Staubli VAL3: Rect10.dtx

public frame fReference = {x=1475.172, y=-187.34, z=-1030, rz=81.293, fatherId=world[0]}
public jointRx jPark = {j3=90, j5=90}
public jointRx jJoint = {j1=-21.01263, j2=66.00245, j3=79.88662, j5=34.11093, j6=162.86516}
public mdesc mNomSpeed = {blend=off}
public mdesc mSpeed[30]
  [0] = {tmax=75, rmax=100, leave=0.1, reach=0.1, blend=cartesian}
  [1] = {tmax=75, rmax=100, leave=0.1, reach=0.1, blend=cartesian}
  [2] = {tmax=75, rmax=100, leave=0.1, reach=0.1, blend=cartesian}
  [3] = {tmax=75, rmax=100, leave=0.1, reach=0.1, blend=cartesian}
  [4] = {tmax=75, rmax=100, leave=0.1, reach=0.1, blend=cartesian}
  [5] = {tmax=75, rmax=100, leave=0.1, reach=0.1, blend=cartesian}
  [6] = {tmax=75, rmax=100, leave=0.1, reach=0.1, blend=cartesian}
  [7] = {tmax=75, rmax=100, leave=0.1, reach=0.1, blend=cartesian}
  [8] = {tmax=75, rmax=100, leave=0.1, reach=0.1, blend=cartesian}
  [9] = {tmax=75, rmax=100, leave=0.1, reach=0.1, blend=cartesian}
  [10] = {tmax=75, rmax=100, leave=0.1, reach=0.1, blend=cartesian}
  [11] = {tmax=75, rmax=100, leave=0.1, reach=0.1, blend=cartesian}
  [12] = {tmax=75, rmax=100, leave=0.1, reach=0.1, blend=cartesian}
  [13] = {tmax=75, rmax=100, leave=0.1, reach=0.1, blend=cartesian}
  [14] = {tmax=75, rmax=100, leave=0.1, reach=0.1, blend=cartesian}
  [15] = {tmax=75, rmax=100, leave=0.1, reach=0.1, blend=cartesian}
  [16] = {tmax=75, rmax=100, leave=0.1, reach=0.1, blend=cartesian}
  [17] = {tmax=75, rmax=100, leave=0.1, reach=0.1, blend=cartesian}
  [18] = {tmax=75, rmax=100, leave=0.1, reach=0.1, blend=cartesian}
  [19] = {tmax=75, rmax=100, leave=0.1, reach=0.1, blend=cartesian}
  [20] = {tmax=75, rmax=100, leave=0.1, reach=0.1, blend=cartesian}
  [21] = {tmax=75, rmax=100, leave=0.1, reach=0.1, blend=cartesian}
  [22] = {tmax=75, rmax=100, leave=0.1, reach=0.1, blend=cartesian}
  [23] = {tmax=75, rmax=100, leave=0.1, reach=0.1, blend=cartesian}
  [24] = {tmax=75, rmax=100, leave=0.1, reach=0.1, blend=cartesian}
  [25] = {tmax=75, rmax=100, leave=0.1, reach=0.1, blend=cartesian}
  [26] = {tmax=75, rmax=100, leave=0.1, reach=0.1, blend=cartesian}
  [27] = {tmax=75, rmax=100, leave=0.1, reach=0.1, blend=cartesian}
  [28] = {tmax=75, rmax=100, leave=0.1, reach=0.1, blend=cartesian}
  [29] = {tmax=75, rmax=100, leave=0.1, reach=0.1, blend=cartesian}
public num nTraj
num nTimeStop
num nTimeStart
num nMode
num nEtat
public pointRx pPoint[740]
  [0] = {x=-372, y=-44, z=100, rx=-180, rz=85.171, shoulder=lefty, elbow=epositive, wrist=wpositive, fatherId=fReference[0]}
  [1] = {x=-372, y=-44, rx=-180, rz=85.171, shoulder=lefty, elbow=epositive, wrist=wpositive, fatherId=fReference[0]}
  [2] = {x=-372, y=-44, rx=-180, rz=85.171, shoulder=lefty, elbow=epositive, wrist=wpositive, fatherId=fReference[0]}
  [3] = {x=-369.477, y=-73.864, rx=-180, rz=75.512, shoulder=lefty, elbow=epositive, wrist=wpositive, fatherId=fReference[0]}
  [4] = {x=-361.979, y=-102.881, rx=-180, rz=65.854, shoulder=lefty, elbow=epositive, wrist=wpositive, fatherId=fReference[0]}
  [5] = {x=-349.719, y=-130.229, rx=180, rz=56.195, shoulder=lefty, elbow=epositive, wrist=wpositive, fatherId=fReference[0]}
  [6] = {x=-333.045, y=-155.133, rx=-180, rz=46.537, shoulder=lefty, elbow=epositive, wrist=wpositive, fatherId=fReference[0]}
  [7] = {x=-312.429, y=-176.886, rx=-180, rz=36.878, shoulder=lefty, elbow=epositive, wrist=wpositive, fatherId=fReference[0]}
  [8] = {x=-288.455, y=-194.872, rx=180, rz=27.22, shoulder=lefty, elbow=epositive, wrist=wpositive, fatherId=fReference[0]}
  [9] = {x=-261.803, y=-208.58, rx=180, rz=17.561, shoulder=lefty, elbow=epositive, wrist=wpositive, fatherId=fReference[0]}
  [10] = {x=-233.23, y=-217.623, rx=180, rz=7.903, shoulder=lefty, elbow=epositive, wrist=wpositive, fatherId=fReference[0]}
  [11] = {x=-203.544, y=-221.744, rx=-180, rz=0.489, shoulder=lefty, elbow=epositive, wrist=wpositive, fatherId=fReference[0]}
  [12] = {x=-173.543, y=-222, rx=180, shoulder=lefty, elbow=epositive, wrist=wpositive, fatherId=fReference[0]}
  [13] = {x=-143.537, y=-222, rx=180, shoulder=lefty, elbow=epositive, wrist=wpositive, fatherId=fReference[0]}
  [14] = {x=-113.531, y=-222, rx=180, shoulder=lefty, elbow=epositive, wrist=wpositive, fatherId=fReference[0]}
  [15] = {x=-83.525, y=-222, rx=180, shoulder=lefty, elbow=epositive, wrist=wpositive, fatherId=fReference[0]}
  [16] = {x=-53.519, y=-222, rx=180, shoulder=lefty, elbow=epositive, wrist=wpositive, fatherId=fReference[0]}
  [17] = {x=-23.513, y=-222, rx=-180, shoulder=lefty, elbow=epositive, wrist=wpositive, fatherId=fReference[0]}
  [18] = {x=6.493, y=-222, rx=-180, shoulder=lefty, elbow=epositive, wrist=wpositive, fatherId=fReference[0]}
  [19] = {x=36.499, y=-222, rx=-180, shoulder=lefty, elbow=epositive, wrist=wpositive, fatherId=fReference[0]}
  [20] = {x=66.504, y=-222, rx=-180, shoulder=lefty, elbow=epositive, wrist=wpositive, fatherId=fReference[0]}
  [21] = {x=96.51, y=-222, rx=180, shoulder=lefty, elbow=epositive, wrist=wpositive, fatherId=fReference[0]}
  [22] = {x=126.516, y=-222, rx=180, shoulder=lefty, elbow=epositive, wrist=wpositive, fatherId=fReference[0]}
  [23] = {x=156.522, y=-222, rx=180, shoulder=lefty, elbow=epositive, wrist=wpositive, fatherId=fReference[0]}
  [24] = {x=186.528, y=-222, rx=-180, rz=-2.723, shoulder=lefty, elbow=epositive, wrist=wpositive, fatherId=fReference[0]}
  [25] = {x=216.474, y=-220.576, rx=180, rz=-12.083, shoulder=lefty, elbow=epositive, wrist=wpositive, fatherId=fReference[0]}
  [26] = {x=245.78, y=-214.302, rx=180, rz=-21.741, shoulder=lefty, elbow=epositive, wrist=wpositive, fatherId=fReference[0]}
  [27] = {x=273.619, y=-203.201, rx=180, rz=-31.4, shoulder=lefty, elbow=epositive, wrist=wpositive, fatherId=fReference[0]}
  [28] = {x=299.2, y=-187.586, rx=180, rz=-41.058, shoulder=lefty, elbow=epositive, wrist=wpositive, fatherId=fReference[0]}
  [29] = {x=321.799, y=-167.901, rx=-180, rz=-50.717, shoulder=lefty, elbow=epositive, wrist=wpositive, fatherId=fReference[0]}
  [30] = {x=340.775, y=-144.703, rx=-180, rz=-60.375, shoulder=lefty, elbow=epositive, wrist=wpositive, fatherId=fReference[0]}
  [31] = {x=355.59, y=-118.65, rx=180, rz=-70.034, shoulder=lefty, elbow=epositive, wrist=wpositive, fatherId=fReference[0]}
  [32] = {x=365.824, y=-90.481, rx=180, rz=-79.692, shoulder=lefty, elbow=epositive, wrist=wpositive, fatherId=fReference[0]}
  [33] = {x=371.187, y=-60.995, rx=180, rz=-88.446, shoulder=lefty, elbow=epositive, wrist=wpositive, fatherId=fReference[0]}
  [34] = {x=372, y=-31.015, rx=180, rz=-90, shoulder=lefty, elbow=epositive, wrist=wpositive, fatherId=fReference[0]}
  [35] = {x=372, y=-1.009, rx=180, rz=-90, shoulder=lefty, elbow=epositive, wrist=wpositive, fatherId=fReference[0]}
  [36] = {x=372, y=28.997, rx=-180, rz=-91.207, shoulder=lefty, elbow=epositive, wrist=wpositive, fatherId=fReference[0]}
  [37] = {x=371.368, y=58.985, rx=-180, rz=-99.658, shoulder=lefty, elbow=epositive, wrist=wpositive, fatherId=fReference[0]}
  [38] = {x=366.34, y=88.531, rx=-180, rz=-109.317, shoulder=lefty, elbow=epositive, wrist=wpositive, fatherId=fReference[0]}
  [39] = {x=356.426, y=116.814, rx=-180, rz=-118.975, shoulder=lefty, elbow=epositive, wrist=wpositive, fatherId=fReference[0]}
  [40] = {x=341.907, y=143.033, rx=-180, rz=-128.634, shoulder=lefty, elbow=epositive, wrist=wpositive, fatherId=fReference[0]}
  [41] = {x=323.195, y=166.444, rx=-180, rz=-138.292, shoulder=lefty, elbow=epositive, wrist=wpositive, fatherId=fReference[0]}
  [42] = {x=300.821, y=186.384, rx=180, rz=-147.951, shoulder=lefty, elbow=epositive, wrist=wpositive, fatherId=fReference[0]}
  [43] = {x=275.418, y=202.288, rx=-180, rz=-157.609, shoulder=lefty, elbow=epositive, wrist=wpositive, fatherId=fReference[0]}
  [44] = {x=247.707, y=213.704, rx=-180, rz=-167.268, shoulder=lefty, elbow=epositive, wrist=wpositive, fatherId=fReference[0]}
  [45] = {x=218.474, y=220.309, rx=-180, rz=-176.767, shoulder=lefty, elbow=epositive, wrist=wpositive, fatherId=fReference[0]}
  [46] = {x=188.546, y=222, rx=-180, rz=180, shoulder=lefty, elbow=epositive, wrist=wpositive, fatherId=fReference[0]}
  [47] = {x=158.54, y=222, rx=-180, rz=180, shoulder=lefty, elbow=epositive, wrist=wpositive, fatherId=fReference[0]}
  [48] = {x=128.534, y=222, rx=-180, rz=180, shoulder=lefty, elbow=epositive, wrist=wpositive, fatherId=fReference[0]}
  [49] = {x=98.528, y=222, rx=-180, rz=180, shoulder=lefty, elbow=epositive, wrist=wpositive, fatherId=fReference[0]}
  [50] = {x=68.522, y=222, rx=-180, rz=180, shoulder=lefty, elbow=epositive, wrist=wpositive, fatherId=fReference[0]}
  [51] = {x=38.516, y=222, rx=-180, rz=180, shoulder=lefty, elbow=epositive, wrist=wpositive, fatherId=fReference[0]}
  [52] = {x=8.51, y=222, rx=-180, rz=180, shoulder=lefty, elbow=epositive, wrist=wpositive, fatherId=fReference[0]}
  [53] = {x=-21.496, y=222, rx=180, rz=180, shoulder=lefty, elbow=epositive, wrist=wpositive, fatherId=fReference[0]}
  [54] = {x=-51.501, y=222, rx=180, rz=180, shoulder=lefty, elbow=epositive, wrist=wpositive, fatherId=fReference[0]}
  [55] = {x=-81.507, y=222, rx=-180, rz=180, shoulder=lefty, elbow=epositive, wrist=wpositive, fatherId=fReference[0]}
  [56] = {x=-111.513, y=222, rx=-180, rz=180, shoulder=lefty, elbow=epositive, wrist=wpositive, fatherId=fReference[0]}
  [57] = {x=-141.519, y=222, rx=180, rz=180, shoulder=lefty, elbow=epositive, wrist=wpositive, fatherId=fReference[0]}
  [58] = {x=-171.525, y=222, rx=180, rz=179.696, shoulder=lefty, elbow=epositive, wrist=wpositive, fatherId=fReference[0]}
  [59] = {x=-201.529, y=221.841, rx=-180, rz=172.747, shoulder=lefty, elbow=epositive, wrist=wpositive, fatherId=fReference[0]}
  [60] = {x=-231.259, y=218.057, rx=-180, rz=163.088, shoulder=lefty, elbow=epositive, wrist=wpositive, fatherId=fReference[0]}
  [61] = {x=-259.934, y=209.338, rx=180, rz=153.43, shoulder=lefty, elbow=epositive, wrist=wpositive, fatherId=fReference[0]}
  [62] = {x=-286.739, y=195.933, rx=180, rz=143.771, shoulder=lefty, elbow=epositive, wrist=wpositive, fatherId=fReference[0]}
  [63] = {x=-310.915, y=178.22, rx=180, rz=134.113, shoulder=lefty, elbow=epositive, wrist=wpositive, fatherId=fReference[0]}
  [64] = {x=-331.776, y=156.702, rx=180, rz=124.454, shoulder=lefty, elbow=epositive, wrist=wpositive, fatherId=fReference[0]}
  [65] = {x=-348.732, y=131.989, rx=180, rz=114.796, shoulder=lefty, elbow=epositive, wrist=wpositive, fatherId=fReference[0]}
  [66] = {x=-361.301, y=104.782, rx=180, rz=105.137, shoulder=lefty, elbow=epositive, wrist=wpositive, fatherId=fReference[0]}
  [67] = {x=-369.127, y=75.851, rx=180, rz=95.479, shoulder=lefty, elbow=epositive, wrist=wpositive, fatherId=fReference[0]}
  [68] = {x=-371.989, y=46.018, rx=180, rz=90.022, shoulder=lefty, elbow=epositive, wrist=wpositive, fatherId=fReference[0]}
  [69] = {x=-372, y=16.012, rx=-180, rz=90, shoulder=lefty, elbow=epositive, wrist=wpositive, fatherId=fReference[0]}
  [70] = {x=-372, y=-13.994, rx=-180, rz=90, shoulder=lefty, elbow=epositive, wrist=wpositive, fatherId=fReference[0]}
  [71] = {x=-372, y=-44, rx=-180, rz=90, shoulder=lefty, elbow=epositive, wrist=wpositive, fatherId=fReference[0]}
  [72] = {x=-372, y=-44, rx=-180, rz=90, shoulder=lefty, elbow=epositive, wrist=wpositive, fatherId=fReference[0]}
  [73] = {x=-372, y=-44, z=100, rx=-180, rz=90, shoulder=lefty, elbow=epositive, wrist=wpositive, fatherId=fReference[0]}
  [74] = {x=-372, y=-44, z=122, rx=-180, rz=90, shoulder=lefty, elbow=epositive, wrist=wpositive, fatherId=fReference[0]}
  [75] = {x=-372, y=-44, z=22, rx=-180, rz=90, shoulder=lefty, elbow=epositive, wrist=wpositive, fatherId=fReference[0]}
  [76] = {x=-372, y=-44, z=22, rx=-180, rz=90, shoulder=lefty, elbow=epositive, wrist=wpositive, fatherId=fReference[0]}
  [77] = {x=-372, y=-13.994, z=22, rx=-180, rz=90, shoulder=lefty, elbow=epositive, wrist=wpositive, fatherId=fReference[0]}
  [78] = {x=-372, y=16.012, z=22, rx=180, rz=90.022, shoulder=lefty, elbow=epositive, wrist=wpositive, fatherId=fReference[0]}
  [79] = {x=-371.989, y=46.018, z=22, rx=180, rz=95.479, shoulder=lefty, elbow=epositive, wrist=wpositive, fatherId=fReference[0]}
  [80] = {x=-369.127, y=75.851, z=22, rx=180, rz=105.137, shoulder=lefty, elbow=epositive, wrist=wpositive, fatherId=fReference[0]}
  [81] = {x=-361.301, y=104.782, z=22, rx=180, rz=114.796, shoulder=lefty, elbow=epositive, wrist=wpositive, fatherId=fReference[0]}
  [82] = {x=-348.732, y=131.989, z=22, rx=180, rz=124.454, shoulder=lefty, elbow=epositive, wrist=wpositive, fatherId=fReference[0]}
  [83] = {x=-331.776, y=156.702, z=22, rx=180, rz=134.113, shoulder=lefty, elbow=epositive, wrist=wpositive, fatherId=fReference[0]}
  [84] = {x=-310.915, y=178.22, z=22, rx=180, rz=143.771, shoulder=lefty, elbow=epositive, wrist=wpositive, fatherId=fReference[0]}
  [85] = {x=-286.739, y=195.933, z=22, rx=180, rz=153.43, shoulder=lefty, elbow=epositive, wrist=wpositive, fatherId=fReference[0]}
  [86] = {x=-259.934, y=209.338, z=22, rx=180, rz=163.088, shoulder=lefty, elbow=epositive, wrist=wpositive, fatherId=fReference[0]}
  [87] = {x=-231.259, y=218.057, z=22, rx=-180, rz=172.747, shoulder=lefty, elbow=epositive, wrist=wpositive, fatherId=fReference[0]}
  [88] = {x=-201.529, y=221.841, z=22, rx=180, rz=179.696, shoulder=lefty, elbow=epositive, wrist=wpositive, fatherId=fReference[0]}
  [89] = {x=-171.525, y=222, z=22, rx=180, rz=180, shoulder=lefty, elbow=epositive, wrist=wpositive, fatherId=fReference[0]}
  [90] = {x=-141.519, y=222, z=22, rx=-180, rz=180, shoulder=lefty, elbow=epositive, wrist=wpositive, fatherId=fReference[0]}
  [91] = {x=-111.513, y=222, z=22, rx=180, rz=180, shoulder=lefty, elbow=epositive, wrist=wpositive, fatherId=fReference[0]}
  [92] = {x=-81.507, y=222, z=22, rx=-180, rz=180, shoulder=lefty, elbow=epositive, wrist=wpositive, fatherId=fReference[0]}
  [93] = {x=-51.501, y=222, z=22, rx=180, rz=180, shoulder=lefty, elbow=epositive, wrist=wpositive, fatherId=fReference[0]}
  [94] = {x=-21.496, y=222, z=22, rx=180, rz=180, shoulder=lefty, elbow=epositive, wrist=wpositive, fatherId=fReference[0]}
  [95] = {x=8.51, y=222, z=22, rx=-180, rz=180, shoulder=lefty, elbow=epositive, wrist=wpositive, fatherId=fReference[0]}
  [96] = {x=38.516, y=222, z=22, rx=180, rz=180, shoulder=lefty, elbow=epositive, wrist=wpositive, fatherId=fReference[0]}
  [97] = {x=68.522, y=222, z=22, rx=180, rz=180, shoulder=lefty, elbow=epositive, wrist=wpositive, fatherId=fReference[0]}
  [98] = {x=98.528, y=222, z=22, rx=-180, rz=180, shoulder=lefty, elbow=epositive, wrist=wpositive, fatherId=fReference[0]}
  [99] = {x=128.534, y=222, z=22, rx=180, rz=180, shoulder=lefty, elbow=epositive, wrist=wpositive, fatherId=fReference[0]}
  [100] = {x=158.54, y=222, z=22, rx=180, rz=180, shoulder=lefty, elbow=epositive, wrist=wpositive, fatherId=fReference[0]}
  [101] = {x=188.546, y=222, z=22, rx=-180, rz=-176.767, shoulder=lefty, elbow=epositive, wrist=wpositive, fatherId=fReference[0]}
  [102] = {x=218.474, y=220.309, z=22, rx=180, rz=-167.268, shoulder=lefty, elbow=epositive, wrist=wpositive, fatherId=fReference[0]}
  [103] = {x=247.707, y=213.704, z=22, rx=-180, rz=-157.609, shoulder=lefty, elbow=epositive, wrist=wpositive, fatherId=fReference[0]}
  [104] = {x=275.418, y=202.288, z=22, rx=180, rz=-147.951, shoulder=lefty, elbow=epositive, wrist=wpositive, fatherId=fReference[0]}
  [105] = {x=300.821, y=186.384, z=22, rx=-180, rz=-138.292, shoulder=lefty, elbow=epositive, wrist=wpositive, fatherId=fReference[0]}
  [106] = {x=323.195, y=166.444, z=22, rx=-180, rz=-128.634, shoulder=lefty, elbow=epositive, wrist=wpositive, fatherId=fReference[0]}
  [107] = {x=341.907, y=143.033, z=22, rx=-180, rz=-118.975, shoulder=lefty, elbow=epositive, wrist=wpositive, fatherId=fReference[0]}
  [108] = {x=356.426, y=116.814, z=22, rx=-180, rz=-109.317, shoulder=lefty, elbow=epositive, wrist=wpositive, fatherId=fReference[0]}
  [109] = {x=366.34, y=88.531, z=22, rx=-180, rz=-99.658, shoulder=lefty, elbow=epositive, wrist=wpositive, fatherId=fReference[0]}
  [110] = {x=371.368, y=58.985, z=22, rx=-180, rz=-91.207, shoulder=lefty, elbow=epositive, wrist=wpositive, fatherId=fReference[0]}
  [111] = {x=372, y=28.997, z=22, rx=180, rz=-90, shoulder=lefty, elbow=epositive, wrist=wpositive, fatherId=fReference[0]}
  [112] = {x=372, y=-1.009, z=22, rx=180, rz=-90, shoulder=lefty, elbow=epositive, wrist=wpositive, fatherId=fReference[0]}
  [113] = {x=372, y=-31.015, z=22, rx=180, rz=-88.446, shoulder=lefty, elbow=epositive, wrist=wpositive, fatherId=fReference[0]}
  [114] = {x=371.187, y=-60.995, z=22, rx=180, rz=-79.692, shoulder=lefty, elbow=epositive, wrist=wpositive, fatherId=fReference[0]}
  [115] = {x=365.824, y=-90.481, z=22, rx=180, rz=-70.034, shoulder=lefty, elbow=epositive, wrist=wpositive, fatherId=fReference[0]}
  [116] = {x=355.59, y=-118.65, z=22, rx=-180, rz=-60.375, shoulder=lefty, elbow=epositive, wrist=wpositive, fatherId=fReference[0]}
  [117] = {x=340.775, y=-144.703, z=22, rx=180, rz=-50.717, shoulder=lefty, elbow=epositive, wrist=wpositive, fatherId=fReference[0]}
  [118] = {x=321.799, y=-167.901, z=22, rx=180, rz=-41.058, shoulder=lefty, elbow=epositive, wrist=wpositive, fatherId=fReference[0]}
  [119] = {x=299.2, y=-187.586, z=22, rx=180, rz=-31.4, shoulder=lefty, elbow=epositive, wrist=wpositive, fatherId=fReference[0]}
  [120] = {x=273.619, y=-203.201, z=22, rx=180, rz=-21.741, shoulder=lefty, elbow=epositive, wrist=wpositive, fatherId=fReference[0]}
  [121] = {x=245.78, y=-214.302, z=22, rx=180, rz=-12.083, shoulder=lefty, elbow=epositive, wrist=wpositive, fatherId=fReference[0]}
  [122] = {x=216.474, y=-220.576, z=22, rx=-180, rz=-2.723, shoulder=lefty, elbow=epositive, wrist=wpositive, fatherId=fReference[0]}
  [123] = {x=186.528, y=-222, z=22, rx=-180, shoulder=lefty, elbow=epositive, wrist=wpositive, fatherId=fReference[0]}
  [124] = {x=156.522, y=-222, z=22, rx=-180, shoulder=lefty, elbow=epositive, wrist=wpositive, fatherId=fReference[0]}
  [125] = {x=126.516, y=-222, z=22, rx=-180, shoulder=lefty, elbow=epositive, wrist=wpositive, fatherId=fReference[0]}
  [126] = {x=96.51, y=-222, z=22, rx=-180, shoulder=lefty, elbow=epositive, wrist=wpositive, fatherId=fReference[0]}
  [127] = {x=66.504, y=-222, z=22, rx=-180, shoulder=lefty, elbow=epositive, wrist=wpositive, fatherId=fReference[0]}
  [128] = {x=36.499, y=-222, z=22, rx=-180, shoulder=lefty, elbow=epositive, wrist=wpositive, fatherId=fReference[0]}
  [129] = {x=6.493, y=-222, z=22, rx=-180, shoulder=lefty, elbow=epositive, wrist=wpositive, fatherId=fReference[0]}
  [130] = {x=-23.513, y=-222, z=22, rx=180, shoulder=lefty, elbow=epositive, wrist=wpositive, fatherId=fReference[0]}
  [131] = {x=-53.519, y=-222, z=22, rx=180, shoulder=lefty, elbow=epositive, wrist=wpositive, fatherId=fReference[0]}
  [132] = {x=-83.525, y=-222, z=22, rx=-180, shoulder=lefty, elbow=epositive, wrist=wpositive, fatherId=fReference[0]}
  [133] = {x=-113.531, y=-222, z=22, rx=180, shoulder=lefty, elbow=epositive, wrist=wpositive, fatherId=fReference[0]}
  [134] = {x=-143.537, y=-222, z=22, rx=-180, shoulder=lefty, elbow=epositive, wrist=wpositive, fatherId=fReference[0]}
  [135] = {x=-173.543, y=-222, z=22, rx=180, rz=0.489, shoulder=lefty, elbow=epositive, wrist=wpositive, fatherId=fReference[0]}
  [136] = {x=-203.544, y=-221.744, z=22, rx=180, rz=7.903, shoulder=lefty, elbow=epositive, wrist=wpositive, fatherId=fReference[0]}
  [137] = {x=-233.23, y=-217.623, z=22, rx=-180, rz=17.561, shoulder=lefty, elbow=epositive, wrist=wpositive, fatherId=fReference[0]}
  [138] = {x=-261.803, y=-208.58, z=22, rx=-180, rz=27.22, shoulder=lefty, elbow=epositive, wrist=wpositive, fatherId=fReference[0]}
  [139] = {x=-288.455, y=-194.872, z=22, rx=-180, rz=36.878, shoulder=lefty, elbow=epositive, wrist=wpositive, fatherId=fReference[0]}
  [140] = {x=-312.429, y=-176.886, z=22, rx=-180, rz=46.537, shoulder=lefty, elbow=epositive, wrist=wpositive, fatherId=fReference[0]}
  [141] = {x=-333.045, y=-155.133, z=22, rx=-180, rz=56.195, shoulder=lefty, elbow=epositive, wrist=wpositive, fatherId=fReference[0]}
  [142] = {x=-349.719, y=-130.229, z=22, rx=180, rz=65.854, shoulder=lefty, elbow=epositive, wrist=wpositive, fatherId=fReference[0]}
  [143] = {x=-361.979, y=-102.881, z=22, rx=-180, rz=75.512, shoulder=lefty, elbow=epositive, wrist=wpositive, fatherId=fReference[0]}
  [144] = {x=-369.477, y=-73.864, z=22, rx=-180, rz=85.171, shoulder=lefty, elbow=epositive, wrist=wpositive, fatherId=fReference[0]}
  [145] = {x=-372, y=-44, z=22, rx=-180, rz=85.171, shoulder=lefty, elbow=epositive, wrist=wpositive, fatherId=fReference[0]}
  [146] = {x=-372, y=-44, z=22, rx=-180, rz=85.171, shoulder=lefty, elbow=epositive, wrist=wpositive, fatherId=fReference[0]}
  [147] = {x=-372, y=-44, z=122, rx=-180, rz=85.171, shoulder=lefty, elbow=epositive, wrist=wpositive, fatherId=fReference[0]}
  [148] = {x=-372, y=-44, z=144, rx=-180, rz=85.171, shoulder=lefty, elbow=epositive, wrist=wpositive, fatherId=fReference[0]}
  [149] = {x=-372, y=-44, z=44, rx=-180, rz=85.171, shoulder=lefty, elbow=epositive, wrist=wpositive, fatherId=fReference[0]}
  [150] = {x=-372, y=-44, z=44, rx=-180, rz=85.171, shoulder=lefty, elbow=epositive, wrist=wpositive, fatherId=fReference[0]}
  [151] = {x=-369.477, y=-73.864, z=44, rx=-180, rz=75.512, shoulder=lefty, elbow=epositive, wrist=wpositive, fatherId=fReference[0]}
  [152] = {x=-361.979, y=-102.881, z=44, rx=-180, rz=65.854, shoulder=lefty, elbow=epositive, wrist=wpositive, fatherId=fReference[0]}
  [153] = {x=-349.719, y=-130.229, z=44, rx=-180, rz=56.195, shoulder=lefty, elbow=epositive, wrist=wpositive, fatherId=fReference[0]}
  [154] = {x=-333.045, y=-155.133, z=44, rx=180, rz=46.537, shoulder=lefty, elbow=epositive, wrist=wpositive, fatherId=fReference[0]}
  [155] = {x=-312.429, y=-176.886, z=44, rx=-180, rz=36.878, shoulder=lefty, elbow=epositive, wrist=wpositive, fatherId=fReference[0]}
  [156] = {x=-288.455, y=-194.872, z=44, rx=180, rz=27.22, shoulder=lefty, elbow=epositive, wrist=wpositive, fatherId=fReference[0]}
  [157] = {x=-261.803, y=-208.58, z=44, rx=-180, rz=17.561, shoulder=lefty, elbow=epositive, wrist=wpositive, fatherId=fReference[0]}
  [158] = {x=-233.23, y=-217.623, z=44, rx=-180, rz=7.903, shoulder=lefty, elbow=epositive, wrist=wpositive, fatherId=fReference[0]}
  [159] = {x=-203.544, y=-221.744, z=44, rx=-180, rz=0.489, shoulder=lefty, elbow=epositive, wrist=wpositive, fatherId=fReference[0]}
  [160] = {x=-173.543, y=-222, z=44, rx=-180, shoulder=lefty, elbow=epositive, wrist=wpositive, fatherId=fReference[0]}
  [161] = {x=-143.537, y=-222, z=44, rx=180, shoulder=lefty, elbow=epositive, wrist=wpositive, fatherId=fReference[0]}
  [162] = {x=-113.531, y=-222, z=44, rx=180, shoulder=lefty, elbow=epositive, wrist=wpositive, fatherId=fReference[0]}
  [163] = {x=-83.525, y=-222, z=44, rx=-180, shoulder=lefty, elbow=epositive, wrist=wpositive, fatherId=fReference[0]}
  [164] = {x=-53.519, y=-222, z=44, rx=180, shoulder=lefty, elbow=epositive, wrist=wpositive, fatherId=fReference[0]}
  [165] = {x=-23.513, y=-222, z=44, rx=180, shoulder=lefty, elbow=epositive, wrist=wpositive, fatherId=fReference[0]}
  [166] = {x=6.493, y=-222, z=44, rx=180, shoulder=lefty, elbow=epositive, wrist=wpositive, fatherId=fReference[0]}
  [167] = {x=36.499, y=-222, z=44, rx=-180, shoulder=lefty, elbow=epositive, wrist=wpositive, fatherId=fReference[0]}
  [168] = {x=66.504, y=-222, z=44, rx=-180, shoulder=lefty, elbow=epositive, wrist=wpositive, fatherId=fReference[0]}
  [169] = {x=96.51, y=-222, z=44, rx=-180, shoulder=lefty, elbow=epositive, wrist=wpositive, fatherId=fReference[0]}
  [170] = {x=126.516, y=-222, z=44, rx=-180, shoulder=lefty, elbow=epositive, wrist=wpositive, fatherId=fReference[0]}
  [171] = {x=156.522, y=-222, z=44, rx=180, shoulder=lefty, elbow=epositive, wrist=wpositive, fatherId=fReference[0]}
  [172] = {x=186.528, y=-222, z=44, rx=-180, rz=-2.723, shoulder=lefty, elbow=epositive, wrist=wpositive, fatherId=fReference[0]}
  [173] = {x=216.474, y=-220.576, z=44, rx=-180, rz=-12.083, shoulder=lefty, elbow=epositive, wrist=wpositive, fatherId=fReference[0]}
  [174] = {x=245.78, y=-214.302, z=44, rx=180, rz=-21.741, shoulder=lefty, elbow=epositive, wrist=wpositive, fatherId=fReference[0]}
  [175] = {x=273.619, y=-203.201, z=44, rx=180, rz=-31.4, shoulder=lefty, elbow=epositive, wrist=wpositive, fatherId=fReference[0]}
  [176] = {x=299.2, y=-187.586, z=44, rx=180, rz=-41.058, shoulder=lefty, elbow=epositive, wrist=wpositive, fatherId=fReference[0]}
  [177] = {x=321.799, y=-167.901, z=44, rx=180, rz=-50.717, shoulder=lefty, elbow=epositive, wrist=wpositive, fatherId=fReference[0]}
  [178] = {x=340.775, y=-144.703, z=44, rx=180, rz=-60.375, shoulder=lefty, elbow=epositive, wrist=wpositive, fatherId=fReference[0]}
  [179] = {x=355.59, y=-118.65, z=44, rx=-180, rz=-70.034, shoulder=lefty, elbow=epositive, wrist=wpositive, fatherId=fReference[0]}
  [180] = {x=365.824, y=-90.481, z=44, rx=180, rz=-79.692, shoulder=lefty, elbow=epositive, wrist=wpositive, fatherId=fReference[0]}
  [181] = {x=371.187, y=-60.995, z=44, rx=180, rz=-88.446, shoulder=lefty, elbow=epositive, wrist=wpositive, fatherId=fReference[0]}
  [182] = {x=372, y=-31.015, z=44, rx=180, rz=-90, shoulder=lefty, elbow=epositive, wrist=wpositive, fatherId=fReference[0]}
  [183] = {x=372, y=-1.009, z=44, rx=180, rz=-90, shoulder=lefty, elbow=epositive, wrist=wpositive, fatherId=fReference[0]}
  [184] = {x=372, y=28.997, z=44, rx=-180, rz=-91.207, shoulder=lefty, elbow=epositive, wrist=wpositive, fatherId=fReference[0]}
  [185] = {x=371.368, y=58.985, z=44, rx=-180, rz=-99.658, shoulder=lefty, elbow=epositive, wrist=wpositive, fatherId=fReference[0]}
  [186] = {x=366.34, y=88.531, z=44, rx=-180, rz=-109.317, shoulder=lefty, elbow=epositive, wrist=wpositive, fatherId=fReference[0]}
  [187] = {x=356.426, y=116.814, z=44, rx=-180, rz=-118.975, shoulder=lefty, elbow=epositive, wrist=wpositive, fatherId=fReference[0]}
  [188] = {x=341.907, y=143.033, z=44, rx=-180, rz=-128.634, shoulder=lefty, elbow=epositive, wrist=wpositive, fatherId=fReference[0]}
  [189] = {x=323.195, y=166.444, z=44, rx=-180, rz=-138.292, shoulder=lefty, elbow=epositive, wrist=wpositive, fatherId=fReference[0]}
  [190] = {x=300.821, y=186.384, z=44, rx=-180, rz=-147.951, shoulder=lefty, elbow=epositive, wrist=wpositive, fatherId=fReference[0]}
  [191] = {x=275.418, y=202.288, z=44, rx=180, rz=-157.609, shoulder=lefty, elbow=epositive, wrist=wpositive, fatherId=fReference[0]}
  [192] = {x=247.707, y=213.704, z=44, rx=-180, rz=-167.268, shoulder=lefty, elbow=epositive, wrist=wpositive, fatherId=fReference[0]}
  [193] = {x=218.474, y=220.309, z=44, rx=-180, rz=-176.767, shoulder=lefty, elbow=epositive, wrist=wpositive, fatherId=fReference[0]}
  [194] = {x=188.546, y=222, z=44, rx=180, rz=180, shoulder=lefty, elbow=epositive, wrist=wpositive, fatherId=fReference[0]}
  [195] = {x=158.54, y=222, z=44, rx=-180, rz=180, shoulder=lefty, elbow=epositive, wrist=wpositive, fatherId=fReference[0]}
  [196] = {x=128.534, y=222, z=44, rx=-180, rz=180, shoulder=lefty, elbow=epositive, wrist=wpositive, fatherId=fReference[0]}
  [197] = {x=98.528, y=222, z=44, rx=180, rz=-180, shoulder=lefty, elbow=epositive, wrist=wpositive, fatherId=fReference[0]}
  [198] = {x=68.522, y=222, z=44, rx=180, rz=-180, shoulder=lefty, elbow=epositive, wrist=wpositive, fatherId=fReference[0]}
  [199] = {x=38.516, y=222, z=44, rx=180, rz=180, shoulder=lefty, elbow=epositive, wrist=wpositive, fatherId=fReference[0]}
  [200] = {x=8.51, y=222, z=44, rx=-180, rz=180, shoulder=lefty, elbow=epositive, wrist=wpositive, fatherId=fReference[0]}
  [201] = {x=-21.496, y=222, z=44, rx=180, rz=180, shoulder=lefty, elbow=epositive, wrist=wpositive, fatherId=fReference[0]}
  [202] = {x=-51.501, y=222, z=44, rx=180, rz=180, shoulder=lefty, elbow=epositive, wrist=wpositive, fatherId=fReference[0]}
  [203] = {x=-81.507, y=222, z=44, rx=-180, rz=180, shoulder=lefty, elbow=epositive, wrist=wpositive, fatherId=fReference[0]}
  [204] = {x=-111.513, y=222, z=44, rx=180, rz=-180, shoulder=lefty, elbow=epositive, wrist=wpositive, fatherId=fReference[0]}
  [205] = {x=-141.519, y=222, z=44, rx=-180, rz=-180, shoulder=lefty, elbow=epositive, wrist=wpositive, fatherId=fReference[0]}
  [206] = {x=-171.525, y=222, z=44, rx=180, rz=179.696, shoulder=lefty, elbow=epositive, wrist=wpositive, fatherId=fReference[0]}
  [207] = {x=-201.529, y=221.841, z=44, rx=-180, rz=172.747, shoulder=lefty, elbow=epositive, wrist=wpositive, fatherId=fReference[0]}
  [208] = {x=-231.259, y=218.057, z=44, rx=-180, rz=163.088, shoulder=lefty, elbow=epositive, wrist=wpositive, fatherId=fReference[0]}
  [209] = {x=-259.934, y=209.338, z=44, rx=-180, rz=153.43, shoulder=lefty, elbow=epositive, wrist=wpositive, fatherId=fReference[0]}
  [210] = {x=-286.739, y=195.933, z=44, rx=-180, rz=143.771, shoulder=lefty, elbow=epositive, wrist=wpositive, fatherId=fReference[0]}
  [211] = {x=-310.915, y=178.22, z=44, rx=180, rz=134.113, shoulder=lefty, elbow=epositive, wrist=wpositive, fatherId=fReference[0]}
  [212] = {x=-331.776, y=156.702, z=44, rx=180, rz=124.454, shoulder=lefty, elbow=epositive, wrist=wpositive, fatherId=fReference[0]}
  [213] = {x=-348.732, y=131.989, z=44, rx=180, rz=114.796, shoulder=lefty, elbow=epositive, wrist=wpositive, fatherId=fReference[0]}
  [214] = {x=-361.301, y=104.782, z=44, rx=180, rz=105.137, shoulder=lefty, elbow=epositive, wrist=wpositive, fatherId=fReference[0]}
  [215] = {x=-369.127, y=75.851, z=44, rx=180, rz=95.479, shoulder=lefty, elbow=epositive, wrist=wpositive, fatherId=fReference[0]}
  [216] = {x=-371.989, y=46.018, z=44, rx=180, rz=90.022, shoulder=lefty, elbow=epositive, wrist=wpositive, fatherId=fReference[0]}
  [217] = {x=-372, y=16.012, z=44, rx=-180, rz=90, shoulder=lefty, elbow=epositive, wrist=wpositive, fatherId=fReference[0]}
  [218] = {x=-372, y=-13.994, z=44, rx=-180, rz=90, shoulder=lefty, elbow=epositive, wrist=wpositive, fatherId=fReference[0]}
  [219] = {x=-372, y=-44, z=44, rx=-180, rz=90, shoulder=lefty, elbow=epositive, wrist=wpositive, fatherId=fReference[0]}
  [220] = {x=-372, y=-44, z=44, rx=-180, rz=90, shoulder=lefty, elbow=epositive, wrist=wpositive, fatherId=fReference[0]}
  [221] = {x=-372, y=-44, z=144, rx=-180, rz=90, shoulder=lefty, elbow=epositive, wrist=wpositive, fatherId=fReference[0]}
  [222] = {x=-372, y=-44, z=166, rx=-180, rz=90, shoulder=lefty, elbow=epositive, wrist=wpositive, fatherId=fReference[0]}
  [223] = {x=-372, y=-44, z=66, rx=-180, rz=90, shoulder=lefty, elbow=epositive, wrist=wpositive, fatherId=fReference[0]}
  [224] = {x=-372, y=-44, z=66, rx=-180, rz=90, shoulder=lefty, elbow=epositive, wrist=wpositive, fatherId=fReference[0]}
  [225] = {x=-372, y=-13.994, z=66, rx=-180, rz=90, shoulder=lefty, elbow=epositive, wrist=wpositive, fatherId=fReference[0]}
  [226] = {x=-372, y=16.012, z=66, rx=180, rz=90.022, shoulder=lefty, elbow=epositive, wrist=wpositive, fatherId=fReference[0]}
  [227] = {x=-371.989, y=46.018, z=66, rx=180, rz=95.479, shoulder=lefty, elbow=epositive, wrist=wpositive, fatherId=fReference[0]}
  [228] = {x=-369.127, y=75.851, z=66, rx=180, rz=105.137, shoulder=lefty, elbow=epositive, wrist=wpositive, fatherId=fReference[0]}
  [229] = {x=-361.301, y=104.782, z=66, rx=180, rz=114.796, shoulder=lefty, elbow=epositive, wrist=wpositive, fatherId=fReference[0]}
  [230] = {x=-348.732, y=131.989, z=66, rx=180, rz=124.454, shoulder=lefty, elbow=epositive, wrist=wpositive, fatherId=fReference[0]}
  [231] = {x=-331.776, y=156.702, z=66, rx=180, rz=134.113, shoulder=lefty, elbow=epositive, wrist=wpositive, fatherId=fReference[0]}
  [232] = {x=-310.915, y=178.22, z=66, rx=-180, rz=143.771, shoulder=lefty, elbow=epositive, wrist=wpositive, fatherId=fReference[0]}
  [233] = {x=-286.739, y=195.933, z=66, rx=180, rz=153.43, shoulder=lefty, elbow=epositive, wrist=wpositive, fatherId=fReference[0]}
  [234] = {x=-259.934, y=209.338, z=66, rx=180, rz=163.088, shoulder=lefty, elbow=epositive, wrist=wpositive, fatherId=fReference[0]}
  [235] = {x=-231.259, y=218.057, z=66, rx=180, rz=172.747, shoulder=lefty, elbow=epositive, wrist=wpositive, fatherId=fReference[0]}
  [236] = {x=-201.529, y=221.841, z=66, rx=-180, rz=179.696, shoulder=lefty, elbow=epositive, wrist=wpositive, fatherId=fReference[0]}
  [237] = {x=-171.525, y=222, z=66, rx=-180, rz=180, shoulder=lefty, elbow=epositive, wrist=wpositive, fatherId=fReference[0]}
  [238] = {x=-141.519, y=222, z=66, rx=180, rz=-180, shoulder=lefty, elbow=epositive, wrist=wpositive, fatherId=fReference[0]}
  [239] = {x=-111.513, y=222, z=66, rx=180, rz=-180, shoulder=lefty, elbow=epositive, wrist=wpositive, fatherId=fReference[0]}
  [240] = {x=-81.507, y=222, z=66, rx=-180, rz=-180, shoulder=lefty, elbow=epositive, wrist=wpositive, fatherId=fReference[0]}
  [241] = {x=-51.501, y=222, z=66, rx=180, rz=180, shoulder=lefty, elbow=epositive, wrist=wpositive, fatherId=fReference[0]}
  [242] = {x=-21.496, y=222, z=66, rx=180, rz=-180, shoulder=lefty, elbow=epositive, wrist=wpositive, fatherId=fReference[0]}
  [243] = {x=8.51, y=222, z=66, rx=-180, rz=-180, shoulder=lefty, elbow=epositive, wrist=wpositive, fatherId=fReference[0]}
  [244] = {x=38.516, y=222, z=66, rx=-180, rz=-180, shoulder=lefty, elbow=epositive, wrist=wpositive, fatherId=fReference[0]}
  [245] = {x=68.522, y=222, z=66, rx=-180, rz=-180, shoulder=lefty, elbow=epositive, wrist=wpositive, fatherId=fReference[0]}
  [246] = {x=98.528, y=222, z=66, rx=180, rz=-180, shoulder=lefty, elbow=epositive, wrist=wpositive, fatherId=fReference[0]}
  [247] = {x=128.534, y=222, z=66, rx=180, rz=180, shoulder=lefty, elbow=epositive, wrist=wpositive, fatherId=fReference[0]}
  [248] = {x=158.54, y=222, z=66, rx=180, rz=-180, shoulder=lefty, elbow=epositive, wrist=wpositive, fatherId=fReference[0]}
  [249] = {x=188.546, y=222, z=66, rx=-180, rz=-176.767, shoulder=lefty, elbow=epositive, wrist=wpositive, fatherId=fReference[0]}
  [250] = {x=218.474, y=220.309, z=66, rx=180, rz=-167.268, shoulder=lefty, elbow=epositive, wrist=wpositive, fatherId=fReference[0]}
  [251] = {x=247.707, y=213.704, z=66, rx=-180, rz=-157.609, shoulder=lefty, elbow=epositive, wrist=wpositive, fatherId=fReference[0]}
  [252] = {x=275.418, y=202.288, z=66, rx=-180, rz=-147.951, shoulder=lefty, elbow=epositive, wrist=wpositive, fatherId=fReference[0]}
  [253] = {x=300.821, y=186.384, z=66, rx=-180, rz=-138.292, shoulder=lefty, elbow=epositive, wrist=wpositive, fatherId=fReference[0]}
  [254] = {x=323.195, y=166.444, z=66, rx=-180, rz=-128.634, shoulder=lefty, elbow=epositive, wrist=wpositive, fatherId=fReference[0]}
  [255] = {x=341.907, y=143.033, z=66, rx=-180, rz=-118.975, shoulder=lefty, elbow=epositive, wrist=wpositive, fatherId=fReference[0]}
  [256] = {x=356.426, y=116.814, z=66, rx=-180, rz=-109.317, shoulder=lefty, elbow=epositive, wrist=wpositive, fatherId=fReference[0]}
  [257] = {x=366.34, y=88.531, z=66, rx=-180, rz=-99.658, shoulder=lefty, elbow=epositive, wrist=wpositive, fatherId=fReference[0]}
  [258] = {x=371.368, y=58.985, z=66, rx=-180, rz=-91.207, shoulder=lefty, elbow=epositive, wrist=wpositive, fatherId=fReference[0]}
  [259] = {x=372, y=28.997, z=66, rx=180, rz=-90, shoulder=lefty, elbow=epositive, wrist=wpositive, fatherId=fReference[0]}
  [260] = {x=372, y=-1.009, z=66, rx=180, rz=-90, shoulder=lefty, elbow=epositive, wrist=wpositive, fatherId=fReference[0]}
  [261] = {x=372, y=-31.015, z=66, rx=180, rz=-88.446, shoulder=lefty, elbow=epositive, wrist=wpositive, fatherId=fReference[0]}
  [262] = {x=371.187, y=-60.995, z=66, rx=180, rz=-79.692, shoulder=lefty, elbow=epositive, wrist=wpositive, fatherId=fReference[0]}
  [263] = {x=365.824, y=-90.481, z=66, rx=180, rz=-70.034, shoulder=lefty, elbow=epositive, wrist=wpositive, fatherId=fReference[0]}
  [264] = {x=355.59, y=-118.65, z=66, rx=180, rz=-60.375, shoulder=lefty, elbow=epositive, wrist=wpositive, fatherId=fReference[0]}
  [265] = {x=340.775, y=-144.703, z=66, rx=180, rz=-50.717, shoulder=lefty, elbow=epositive, wrist=wpositive, fatherId=fReference[0]}
  [266] = {x=321.799, y=-167.901, z=66, rx=180, rz=-41.058, shoulder=lefty, elbow=epositive, wrist=wpositive, fatherId=fReference[0]}
  [267] = {x=299.2, y=-187.586, z=66, rx=180, rz=-31.4, shoulder=lefty, elbow=epositive, wrist=wpositive, fatherId=fReference[0]}
  [268] = {x=273.619, y=-203.201, z=66, rx=180, rz=-21.741, shoulder=lefty, elbow=epositive, wrist=wpositive, fatherId=fReference[0]}
  [269] = {x=245.78, y=-214.302, z=66, rx=180, rz=-12.083, shoulder=lefty, elbow=epositive, wrist=wpositive, fatherId=fReference[0]}
  [270] = {x=216.474, y=-220.576, z=66, rx=-180, rz=-2.723, shoulder=lefty, elbow=epositive, wrist=wpositive, fatherId=fReference[0]}
  [271] = {x=186.528, y=-222, z=66, rx=-180, shoulder=lefty, elbow=epositive, wrist=wpositive, fatherId=fReference[0]}
  [272] = {x=156.522, y=-222, z=66, rx=180, shoulder=lefty, elbow=epositive, wrist=wpositive, fatherId=fReference[0]}
  [273] = {x=126.516, y=-222, z=66, rx=180, shoulder=lefty, elbow=epositive, wrist=wpositive, fatherId=fReference[0]}
  [274] = {x=96.51, y=-222, z=66, rx=180, shoulder=lefty, elbow=epositive, wrist=wpositive, fatherId=fReference[0]}
  [275] = {x=66.504, y=-222, z=66, rx=-180, shoulder=lefty, elbow=epositive, wrist=wpositive, fatherId=fReference[0]}
  [276] = {x=36.499, y=-222, z=66, rx=-180, shoulder=lefty, elbow=epositive, wrist=wpositive, fatherId=fReference[0]}
  [277] = {x=6.493, y=-222, z=66, rx=-180, shoulder=lefty, elbow=epositive, wrist=wpositive, fatherId=fReference[0]}
  [278] = {x=-23.513, y=-222, z=66, rx=-180, shoulder=lefty, elbow=epositive, wrist=wpositive, fatherId=fReference[0]}
  [279] = {x=-53.519, y=-222, z=66, rx=180, shoulder=lefty, elbow=epositive, wrist=wpositive, fatherId=fReference[0]}
  [280] = {x=-83.525, y=-222, z=66, rx=-180, shoulder=lefty, elbow=epositive, wrist=wpositive, fatherId=fReference[0]}
  [281] = {x=-113.531, y=-222, z=66, rx=-180, shoulder=lefty, elbow=epositive, wrist=wpositive, fatherId=fReference[0]}
  [282] = {x=-143.537, y=-222, z=66, rx=-180, shoulder=lefty, elbow=epositive, wrist=wpositive, fatherId=fReference[0]}
  [283] = {x=-173.543, y=-222, z=66, rx=180, rz=0.489, shoulder=lefty, elbow=epositive, wrist=wpositive, fatherId=fReference[0]}
  [284] = {x=-203.544, y=-221.744, z=66, rx=180, rz=7.903, shoulder=lefty, elbow=epositive, wrist=wpositive, fatherId=fReference[0]}
  [285] = {x=-233.23, y=-217.623, z=66, rx=-180, rz=17.561, shoulder=lefty, elbow=epositive, wrist=wpositive, fatherId=fReference[0]}
  [286] = {x=-261.803, y=-208.58, z=66, rx=180, rz=27.22, shoulder=lefty, elbow=epositive, wrist=wpositive, fatherId=fReference[0]}
  [287] = {x=-288.455, y=-194.872, z=66, rx=-180, rz=36.878, shoulder=lefty, elbow=epositive, wrist=wpositive, fatherId=fReference[0]}
  [288] = {x=-312.429, y=-176.886, z=66, rx=-180, rz=46.537, shoulder=lefty, elbow=epositive, wrist=wpositive, fatherId=fReference[0]}
  [289] = {x=-333.045, y=-155.133, z=66, rx=-180, rz=56.195, shoulder=lefty, elbow=epositive, wrist=wpositive, fatherId=fReference[0]}
  [290] = {x=-349.719, y=-130.229, z=66, rx=-180, rz=65.854, shoulder=lefty, elbow=epositive, wrist=wpositive, fatherId=fReference[0]}
  [291] = {x=-361.979, y=-102.881, z=66, rx=-180, rz=75.512, shoulder=lefty, elbow=epositive, wrist=wpositive, fatherId=fReference[0]}
  [292] = {x=-369.477, y=-73.864, z=66, rx=-180, rz=85.171, shoulder=lefty, elbow=epositive, wrist=wpositive, fatherId=fReference[0]}
  [293] = {x=-372, y=-44, z=66, rx=-180, rz=85.171, shoulder=lefty, elbow=epositive, wrist=wpositive, fatherId=fReference[0]}
  [294] = {x=-372, y=-44, z=66, rx=-180, rz=85.171, shoulder=lefty, elbow=epositive, wrist=wpositive, fatherId=fReference[0]}
  [295] = {x=-372, y=-44, z=166, rx=-180, rz=85.171, shoulder=lefty, elbow=epositive, wrist=wpositive, fatherId=fReference[0]}
  [296] = {x=-372, y=-44, z=188, rx=-180, rz=85.171, shoulder=lefty, elbow=epositive, wrist=wpositive, fatherId=fReference[0]}
  [297] = {x=-372, y=-44, z=88, rx=-180, rz=85.171, shoulder=lefty, elbow=epositive, wrist=wpositive, fatherId=fReference[0]}
  [298] = {x=-372, y=-44, z=88, rx=-180, rz=85.171, shoulder=lefty, elbow=epositive, wrist=wpositive, fatherId=fReference[0]}
  [299] = {x=-369.477, y=-73.864, z=88, rx=-180, rz=75.512, shoulder=lefty, elbow=epositive, wrist=wpositive, fatherId=fReference[0]}
  [300] = {x=-361.979, y=-102.881, z=88, rx=-180, rz=65.854, shoulder=lefty, elbow=epositive, wrist=wpositive, fatherId=fReference[0]}
  [301] = {x=-349.719, y=-130.229, z=88, rx=-180, rz=56.195, shoulder=lefty, elbow=epositive, wrist=wpositive, fatherId=fReference[0]}
  [302] = {x=-333.045, y=-155.133, z=88, rx=-180, rz=46.537, shoulder=lefty, elbow=epositive, wrist=wpositive, fatherId=fReference[0]}
  [303] = {x=-312.429, y=-176.886, z=88, rx=-180, rz=36.878, shoulder=lefty, elbow=epositive, wrist=wpositive, fatherId=fReference[0]}
  [304] = {x=-288.455, y=-194.872, z=88, rx=-180, rz=27.22, shoulder=lefty, elbow=epositive, wrist=wpositive, fatherId=fReference[0]}
  [305] = {x=-261.803, y=-208.58, z=88, rx=-180, rz=17.561, shoulder=lefty, elbow=epositive, wrist=wpositive, fatherId=fReference[0]}
  [306] = {x=-233.23, y=-217.623, z=88, rx=180, rz=7.903, shoulder=lefty, elbow=epositive, wrist=wpositive, fatherId=fReference[0]}
  [307] = {x=-203.544, y=-221.744, z=88, rx=-180, rz=0.489, shoulder=lefty, elbow=epositive, wrist=wpositive, fatherId=fReference[0]}
  [308] = {x=-173.543, y=-222, z=88, rx=180, shoulder=lefty, elbow=epositive, wrist=wpositive, fatherId=fReference[0]}
  [309] = {x=-143.537, y=-222, z=88, rx=-180, shoulder=lefty, elbow=epositive, wrist=wpositive, fatherId=fReference[0]}
  [310] = {x=-113.531, y=-222, z=88, rx=-180, shoulder=lefty, elbow=epositive, wrist=wpositive, fatherId=fReference[0]}
  [311] = {x=-83.525, y=-222, z=88, rx=180, shoulder=lefty, elbow=epositive, wrist=wpositive, fatherId=fReference[0]}
  [312] = {x=-53.519, y=-222, z=88, rx=-180, shoulder=lefty, elbow=epositive, wrist=wpositive, fatherId=fReference[0]}
  [313] = {x=-23.513, y=-222, z=88, rx=-180, shoulder=lefty, elbow=epositive, wrist=wpositive, fatherId=fReference[0]}
  [314] = {x=6.493, y=-222, z=88, rx=-180, shoulder=lefty, elbow=epositive, wrist=wpositive, fatherId=fReference[0]}
  [315] = {x=36.499, y=-222, z=88, rx=-180, shoulder=lefty, elbow=epositive, wrist=wpositive, fatherId=fReference[0]}
  [316] = {x=66.504, y=-222, z=88, rx=-180, shoulder=lefty, elbow=epositive, wrist=wpositive, fatherId=fReference[0]}
  [317] = {x=96.51, y=-222, z=88, rx=-180, shoulder=lefty, elbow=epositive, wrist=wpositive, fatherId=fReference[0]}
  [318] = {x=126.516, y=-222, z=88, rx=-180, shoulder=lefty, elbow=epositive, wrist=wpositive, fatherId=fReference[0]}
  [319] = {x=156.522, y=-222, z=88, rx=-180, shoulder=lefty, elbow=epositive, wrist=wpositive, fatherId=fReference[0]}
  [320] = {x=186.528, y=-222, z=88, rx=180, rz=-2.723, shoulder=lefty, elbow=epositive, wrist=wpositive, fatherId=fReference[0]}
  [321] = {x=216.474, y=-220.576, z=88, rx=180, rz=-12.083, shoulder=lefty, elbow=epositive, wrist=wpositive, fatherId=fReference[0]}
  [322] = {x=245.78, y=-214.302, z=88, rx=180, rz=-21.741, shoulder=lefty, elbow=epositive, wrist=wpositive, fatherId=fReference[0]}
  [323] = {x=273.619, y=-203.201, z=88, rx=180, rz=-31.4, shoulder=lefty, elbow=epositive, wrist=wpositive, fatherId=fReference[0]}
  [324] = {x=299.2, y=-187.586, z=88, rx=-180, rz=-41.058, shoulder=lefty, elbow=epositive, wrist=wpositive, fatherId=fReference[0]}
  [325] = {x=321.799, y=-167.901, z=88, rx=180, rz=-50.717, shoulder=lefty, elbow=epositive, wrist=wpositive, fatherId=fReference[0]}
  [326] = {x=340.775, y=-144.703, z=88, rx=-180, rz=-60.375, shoulder=lefty, elbow=epositive, wrist=wpositive, fatherId=fReference[0]}
  [327] = {x=355.59, y=-118.65, z=88, rx=180, rz=-70.034, shoulder=lefty, elbow=epositive, wrist=wpositive, fatherId=fReference[0]}
  [328] = {x=365.824, y=-90.481, z=88, rx=180, rz=-79.692, shoulder=lefty, elbow=epositive, wrist=wpositive, fatherId=fReference[0]}
  [329] = {x=371.187, y=-60.995, z=88, rx=180, rz=-88.446, shoulder=lefty, elbow=epositive, wrist=wpositive, fatherId=fReference[0]}
  [330] = {x=372, y=-31.015, z=88, rx=180, rz=-90, shoulder=lefty, elbow=epositive, wrist=wpositive, fatherId=fReference[0]}
  [331] = {x=372, y=-1.009, z=88, rx=180, rz=-90, shoulder=lefty, elbow=epositive, wrist=wpositive, fatherId=fReference[0]}
  [332] = {x=372, y=28.997, z=88, rx=-180, rz=-91.207, shoulder=lefty, elbow=epositive, wrist=wpositive, fatherId=fReference[0]}
  [333] = {x=371.368, y=58.985, z=88, rx=-180, rz=-99.658, shoulder=lefty, elbow=epositive, wrist=wpositive, fatherId=fReference[0]}
  [334] = {x=366.34, y=88.531, z=88, rx=-180, rz=-109.317, shoulder=lefty, elbow=epositive, wrist=wpositive, fatherId=fReference[0]}
  [335] = {x=356.426, y=116.814, z=88, rx=-180, rz=-118.975, shoulder=lefty, elbow=epositive, wrist=wpositive, fatherId=fReference[0]}
  [336] = {x=341.907, y=143.033, z=88, rx=-180, rz=-128.634, shoulder=lefty, elbow=epositive, wrist=wpositive, fatherId=fReference[0]}
  [337] = {x=323.195, y=166.444, z=88, rx=-180, rz=-138.292, shoulder=lefty, elbow=epositive, wrist=wpositive, fatherId=fReference[0]}
  [338] = {x=300.821, y=186.384, z=88, rx=-180, rz=-147.951, shoulder=lefty, elbow=epositive, wrist=wpositive, fatherId=fReference[0]}
  [339] = {x=275.418, y=202.288, z=88, rx=-180, rz=-157.609, shoulder=lefty, elbow=epositive, wrist=wpositive, fatherId=fReference[0]}
  [340] = {x=247.707, y=213.704, z=88, rx=-180, rz=-167.268, shoulder=lefty, elbow=epositive, wrist=wpositive, fatherId=fReference[0]}
  [341] = {x=218.474, y=220.309, z=88, rx=-180, rz=-176.767, shoulder=lefty, elbow=epositive, wrist=wpositive, fatherId=fReference[0]}
  [342] = {x=188.546, y=222, z=88, rx=180, rz=180, shoulder=lefty, elbow=epositive, wrist=wpositive, fatherId=fReference[0]}
  [343] = {x=158.54, y=222, z=88, rx=-180, rz=-180, shoulder=lefty, elbow=epositive, wrist=wpositive, fatherId=fReference[0]}
  [344] = {x=128.534, y=222, z=88, rx=180, rz=-180, shoulder=lefty, elbow=epositive, wrist=wpositive, fatherId=fReference[0]}
  [345] = {x=98.528, y=222, z=88, rx=-180, rz=-180, shoulder=lefty, elbow=epositive, wrist=wpositive, fatherId=fReference[0]}
  [346] = {x=68.522, y=222, z=88, rx=-180, rz=-180, shoulder=lefty, elbow=epositive, wrist=wpositive, fatherId=fReference[0]}
  [347] = {x=38.516, y=222, z=88, rx=180, rz=-180, shoulder=lefty, elbow=epositive, wrist=wpositive, fatherId=fReference[0]}
  [348] = {x=8.51, y=222, z=88, rx=-180, rz=-180, shoulder=lefty, elbow=epositive, wrist=wpositive, fatherId=fReference[0]}
  [349] = {x=-21.496, y=222, z=88, rx=180, rz=-180, shoulder=lefty, elbow=epositive, wrist=wpositive, fatherId=fReference[0]}
  [350] = {x=-51.501, y=222, z=88, rx=180, rz=180, shoulder=lefty, elbow=epositive, wrist=wpositive, fatherId=fReference[0]}
  [351] = {x=-81.507, y=222, z=88, rx=180, rz=-180, shoulder=lefty, elbow=epositive, wrist=wpositive, fatherId=fReference[0]}
  [352] = {x=-111.513, y=222, z=88, rx=180, rz=-180, shoulder=lefty, elbow=epositive, wrist=wpositive, fatherId=fReference[0]}
  [353] = {x=-141.519, y=222, z=88, rx=180, rz=-180, shoulder=lefty, elbow=epositive, wrist=wpositive, fatherId=fReference[0]}
  [354] = {x=-171.525, y=222, z=88, rx=180, rz=179.696, shoulder=lefty, elbow=epositive, wrist=wpositive, fatherId=fReference[0]}
  [355] = {x=-201.529, y=221.841, z=88, rx=180, rz=172.747, shoulder=lefty, elbow=epositive, wrist=wpositive, fatherId=fReference[0]}
  [356] = {x=-231.259, y=218.057, z=88, rx=-180, rz=163.088, shoulder=lefty, elbow=epositive, wrist=wpositive, fatherId=fReference[0]}
  [357] = {x=-259.934, y=209.338, z=88, rx=180, rz=153.43, shoulder=lefty, elbow=epositive, wrist=wpositive, fatherId=fReference[0]}
  [358] = {x=-286.739, y=195.933, z=88, rx=180, rz=143.771, shoulder=lefty, elbow=epositive, wrist=wpositive, fatherId=fReference[0]}
  [359] = {x=-310.915, y=178.22, z=88, rx=180, rz=134.113, shoulder=lefty, elbow=epositive, wrist=wpositive, fatherId=fReference[0]}
  [360] = {x=-331.776, y=156.702, z=88, rx=180, rz=124.454, shoulder=lefty, elbow=epositive, wrist=wpositive, fatherId=fReference[0]}
  [361] = {x=-348.732, y=131.989, z=88, rx=180, rz=114.796, shoulder=lefty, elbow=epositive, wrist=wpositive, fatherId=fReference[0]}
  [362] = {x=-361.301, y=104.782, z=88, rx=180, rz=105.137, shoulder=lefty, elbow=epositive, wrist=wpositive, fatherId=fReference[0]}
  [363] = {x=-369.127, y=75.851, z=88, rx=180, rz=95.479, shoulder=lefty, elbow=epositive, wrist=wpositive, fatherId=fReference[0]}
  [364] = {x=-371.989, y=46.018, z=88, rx=180, rz=90.022, shoulder=lefty, elbow=epositive, wrist=wpositive, fatherId=fReference[0]}
  [365] = {x=-372, y=16.012, z=88, rx=-180, rz=90, shoulder=lefty, elbow=epositive, wrist=wpositive, fatherId=fReference[0]}
  [366] = {x=-372, y=-13.994, z=88, rx=-180, rz=90, shoulder=lefty, elbow=epositive, wrist=wpositive, fatherId=fReference[0]}
  [367] = {x=-372, y=-44, z=88, rx=-180, rz=90, shoulder=lefty, elbow=epositive, wrist=wpositive, fatherId=fReference[0]}
  [368] = {x=-372, y=-44, z=88, rx=-180, rz=90, shoulder=lefty, elbow=epositive, wrist=wpositive, fatherId=fReference[0]}
  [369] = {x=-372, y=-44, z=188, rx=-180, rz=90, shoulder=lefty, elbow=epositive, wrist=wpositive, fatherId=fReference[0]}
  [370] = {x=-372, y=-44, z=210, rx=-180, rz=90, shoulder=lefty, elbow=epositive, wrist=wpositive, fatherId=fReference[0]}
  [371] = {x=-372, y=-44, z=110, rx=-180, rz=90, shoulder=lefty, elbow=epositive, wrist=wpositive, fatherId=fReference[0]}
  [372] = {x=-372, y=-44, z=110, rx=-180, rz=90, shoulder=lefty, elbow=epositive, wrist=wpositive, fatherId=fReference[0]}
  [373] = {x=-372, y=-13.994, z=110, rx=-180, rz=90, shoulder=lefty, elbow=epositive, wrist=wpositive, fatherId=fReference[0]}
  [374] = {x=-372, y=16.012, z=110, rx=180, rz=90.022, shoulder=lefty, elbow=epositive, wrist=wpositive, fatherId=fReference[0]}
  [375] = {x=-371.989, y=46.018, z=110, rx=180, rz=95.479, shoulder=lefty, elbow=epositive, wrist=wpositive, fatherId=fReference[0]}
  [376] = {x=-369.127, y=75.851, z=110, rx=180, rz=105.137, shoulder=lefty, elbow=epositive, wrist=wpositive, fatherId=fReference[0]}
  [377] = {x=-361.301, y=104.782, z=110, rx=180, rz=114.796, shoulder=lefty, elbow=epositive, wrist=wpositive, fatherId=fReference[0]}
  [378] = {x=-348.732, y=131.989, z=110, rx=-180, rz=124.454, shoulder=lefty, elbow=epositive, wrist=wpositive, fatherId=fReference[0]}
  [379] = {x=-331.776, y=156.702, z=110, rx=180, rz=134.113, shoulder=lefty, elbow=epositive, wrist=wpositive, fatherId=fReference[0]}
  [380] = {x=-310.915, y=178.22, z=110, rx=180, rz=143.771, shoulder=lefty, elbow=epositive, wrist=wpositive, fatherId=fReference[0]}
  [381] = {x=-286.739, y=195.933, z=110, rx=-180, rz=153.43, shoulder=lefty, elbow=epositive, wrist=wpositive, fatherId=fReference[0]}
  [382] = {x=-259.934, y=209.338, z=110, rx=180, rz=163.088, shoulder=lefty, elbow=epositive, wrist=wpositive, fatherId=fReference[0]}
  [383] = {x=-231.259, y=218.057, z=110, rx=-180, rz=172.747, shoulder=lefty, elbow=epositive, wrist=wpositive, fatherId=fReference[0]}
  [384] = {x=-201.529, y=221.841, z=110, rx=180, rz=179.696, shoulder=lefty, elbow=epositive, wrist=wpositive, fatherId=fReference[0]}
  [385] = {x=-171.525, y=222, z=110, rx=-180, rz=180, shoulder=lefty, elbow=epositive, wrist=wpositive, fatherId=fReference[0]}
  [386] = {x=-141.519, y=222, z=110, rx=180, rz=-180, shoulder=lefty, elbow=epositive, wrist=wpositive, fatherId=fReference[0]}
  [387] = {x=-111.513, y=222, z=110, rx=-180, rz=-180, shoulder=lefty, elbow=epositive, wrist=wpositive, fatherId=fReference[0]}
  [388] = {x=-81.507, y=222, z=110, rx=-180, rz=-180, shoulder=lefty, elbow=epositive, wrist=wpositive, fatherId=fReference[0]}
  [389] = {x=-51.501, y=222, z=110, rx=180, rz=-180, shoulder=lefty, elbow=epositive, wrist=wpositive, fatherId=fReference[0]}
  [390] = {x=-21.496, y=222, z=110, rx=-180, rz=-180, shoulder=lefty, elbow=epositive, wrist=wpositive, fatherId=fReference[0]}
  [391] = {x=8.51, y=222, z=110, rx=-180, rz=-180, shoulder=lefty, elbow=epositive, wrist=wpositive, fatherId=fReference[0]}
  [392] = {x=38.516, y=222, z=110, rx=-180, rz=-180, shoulder=lefty, elbow=epositive, wrist=wpositive, fatherId=fReference[0]}
  [393] = {x=68.522, y=222, z=110, rx=180, rz=-180, shoulder=lefty, elbow=epositive, wrist=wpositive, fatherId=fReference[0]}
  [394] = {x=98.528, y=222, z=110, rx=-180, rz=-180, shoulder=lefty, elbow=epositive, wrist=wpositive, fatherId=fReference[0]}
  [395] = {x=128.534, y=222, z=110, rx=180, rz=-180, shoulder=lefty, elbow=epositive, wrist=wpositive, fatherId=fReference[0]}
  [396] = {x=158.54, y=222, z=110, rx=180, rz=-180, shoulder=lefty, elbow=epositive, wrist=wpositive, fatherId=fReference[0]}
  [397] = {x=188.546, y=222, z=110, rx=-180, rz=-176.767, shoulder=lefty, elbow=epositive, wrist=wpositive, fatherId=fReference[0]}
  [398] = {x=218.474, y=220.309, z=110, rx=-180, rz=-167.268, shoulder=lefty, elbow=epositive, wrist=wpositive, fatherId=fReference[0]}
  [399] = {x=247.707, y=213.704, z=110, rx=-180, rz=-157.609, shoulder=lefty, elbow=epositive, wrist=wpositive, fatherId=fReference[0]}
  [400] = {x=275.418, y=202.288, z=110, rx=-180, rz=-147.951, shoulder=lefty, elbow=epositive, wrist=wpositive, fatherId=fReference[0]}
  [401] = {x=300.821, y=186.384, z=110, rx=180, rz=-138.292, shoulder=lefty, elbow=epositive, wrist=wpositive, fatherId=fReference[0]}
  [402] = {x=323.195, y=166.444, z=110, rx=-180, rz=-128.634, shoulder=lefty, elbow=epositive, wrist=wpositive, fatherId=fReference[0]}
  [403] = {x=341.907, y=143.033, z=110, rx=-180, rz=-118.975, shoulder=lefty, elbow=epositive, wrist=wpositive, fatherId=fReference[0]}
  [404] = {x=356.426, y=116.814, z=110, rx=-180, rz=-109.317, shoulder=lefty, elbow=epositive, wrist=wpositive, fatherId=fReference[0]}
  [405] = {x=366.34, y=88.531, z=110, rx=-180, rz=-99.658, shoulder=lefty, elbow=epositive, wrist=wpositive, fatherId=fReference[0]}
  [406] = {x=371.368, y=58.985, z=110, rx=-180, rz=-91.207, shoulder=lefty, elbow=epositive, wrist=wpositive, fatherId=fReference[0]}
  [407] = {x=372, y=28.997, z=110, rx=180, rz=-90, shoulder=lefty, elbow=epositive, wrist=wpositive, fatherId=fReference[0]}
  [408] = {x=372, y=-1.009, z=110, rx=180, rz=-90, shoulder=lefty, elbow=epositive, wrist=wpositive, fatherId=fReference[0]}
  [409] = {x=372, y=-31.015, z=110, rx=180, rz=-88.446, shoulder=lefty, elbow=epositive, wrist=wpositive, fatherId=fReference[0]}
  [410] = {x=371.187, y=-60.995, z=110, rx=180, rz=-79.692, shoulder=lefty, elbow=epositive, wrist=wpositive, fatherId=fReference[0]}
  [411] = {x=365.824, y=-90.481, z=110, rx=180, rz=-70.034, shoulder=lefty, elbow=epositive, wrist=wpositive, fatherId=fReference[0]}
  [412] = {x=355.59, y=-118.65, z=110, rx=-180, rz=-60.375, shoulder=lefty, elbow=epositive, wrist=wpositive, fatherId=fReference[0]}
  [413] = {x=340.775, y=-144.703, z=110, rx=180, rz=-50.717, shoulder=lefty, elbow=epositive, wrist=wpositive, fatherId=fReference[0]}
  [414] = {x=321.799, y=-167.901, z=110, rx=-180, rz=-41.058, shoulder=lefty, elbow=epositive, wrist=wpositive, fatherId=fReference[0]}
  [415] = {x=299.2, y=-187.586, z=110, rx=-180, rz=-31.4, shoulder=lefty, elbow=epositive, wrist=wpositive, fatherId=fReference[0]}
  [416] = {x=273.619, y=-203.201, z=110, rx=-180, rz=-21.741, shoulder=lefty, elbow=epositive, wrist=wpositive, fatherId=fReference[0]}
  [417] = {x=245.78, y=-214.302, z=110, rx=-180, rz=-12.083, shoulder=lefty, elbow=epositive, wrist=wpositive, fatherId=fReference[0]}
  [418] = {x=216.474, y=-220.576, z=110, rx=180, rz=-2.723, shoulder=lefty, elbow=epositive, wrist=wpositive, fatherId=fReference[0]}
  [419] = {x=186.528, y=-222, z=110, rx=-180, shoulder=lefty, elbow=epositive, wrist=wpositive, fatherId=fReference[0]}
  [420] = {x=156.522, y=-222, z=110, rx=180, shoulder=lefty, elbow=epositive, wrist=wpositive, fatherId=fReference[0]}
  [421] = {x=126.516, y=-222, z=110, rx=180, shoulder=lefty, elbow=epositive, wrist=wpositive, fatherId=fReference[0]}
  [422] = {x=96.51, y=-222, z=110, rx=-180, shoulder=lefty, elbow=epositive, wrist=wpositive, fatherId=fReference[0]}
  [423] = {x=66.504, y=-222, z=110, rx=180, shoulder=lefty, elbow=epositive, wrist=wpositive, fatherId=fReference[0]}
  [424] = {x=36.499, y=-222, z=110, rx=-180, shoulder=lefty, elbow=epositive, wrist=wpositive, fatherId=fReference[0]}
  [425] = {x=6.493, y=-222, z=110, rx=-180, shoulder=lefty, elbow=epositive, wrist=wpositive, fatherId=fReference[0]}
  [426] = {x=-23.513, y=-222, z=110, rx=180, shoulder=lefty, elbow=epositive, wrist=wpositive, fatherId=fReference[0]}
  [427] = {x=-53.519, y=-222, z=110, rx=180, shoulder=lefty, elbow=epositive, wrist=wpositive, fatherId=fReference[0]}
  [428] = {x=-83.525, y=-222, z=110, rx=-180, shoulder=lefty, elbow=epositive, wrist=wpositive, fatherId=fReference[0]}
  [429] = {x=-113.531, y=-222, z=110, rx=-180, shoulder=lefty, elbow=epositive, wrist=wpositive, fatherId=fReference[0]}
  [430] = {x=-143.537, y=-222, z=110, rx=180, shoulder=lefty, elbow=epositive, wrist=wpositive, fatherId=fReference[0]}
  [431] = {x=-173.543, y=-222, z=110, rx=180, rz=0.489, shoulder=lefty, elbow=epositive, wrist=wpositive, fatherId=fReference[0]}
  [432] = {x=-203.544, y=-221.744, z=110, rx=180, rz=7.903, shoulder=lefty, elbow=epositive, wrist=wpositive, fatherId=fReference[0]}
  [433] = {x=-233.23, y=-217.623, z=110, rx=-180, rz=17.561, shoulder=lefty, elbow=epositive, wrist=wpositive, fatherId=fReference[0]}
  [434] = {x=-261.803, y=-208.58, z=110, rx=-180, rz=27.22, shoulder=lefty, elbow=epositive, wrist=wpositive, fatherId=fReference[0]}
  [435] = {x=-288.455, y=-194.872, z=110, rx=-180, rz=36.878, shoulder=lefty, elbow=epositive, wrist=wpositive, fatherId=fReference[0]}
  [436] = {x=-312.429, y=-176.886, z=110, rx=-180, rz=46.537, shoulder=lefty, elbow=epositive, wrist=wpositive, fatherId=fReference[0]}
  [437] = {x=-333.045, y=-155.133, z=110, rx=-180, rz=56.195, shoulder=lefty, elbow=epositive, wrist=wpositive, fatherId=fReference[0]}
  [438] = {x=-349.719, y=-130.229, z=110, rx=-180, rz=65.854, shoulder=lefty, elbow=epositive, wrist=wpositive, fatherId=fReference[0]}
  [439] = {x=-361.979, y=-102.881, z=110, rx=-180, rz=75.512, shoulder=lefty, elbow=epositive, wrist=wpositive, fatherId=fReference[0]}
  [440] = {x=-369.477, y=-73.864, z=110, rx=-180, rz=85.171, shoulder=lefty, elbow=epositive, wrist=wpositive, fatherId=fReference[0]}
  [441] = {x=-372, y=-44, z=110, rx=-180, rz=85.171, shoulder=lefty, elbow=epositive, wrist=wpositive, fatherId=fReference[0]}
  [442] = {x=-372, y=-44, z=110, rx=-180, rz=85.171, shoulder=lefty, elbow=epositive, wrist=wpositive, fatherId=fReference[0]}
  [443] = {x=-372, y=-44, z=210, rx=-180, rz=85.171, shoulder=lefty, elbow=epositive, wrist=wpositive, fatherId=fReference[0]}
  [444] = {x=-372, y=-44, z=232, rx=-180, rz=85.171, shoulder=lefty, elbow=epositive, wrist=wpositive, fatherId=fReference[0]}
  [445] = {x=-372, y=-44, z=132, rx=-180, rz=85.171, shoulder=lefty, elbow=epositive, wrist=wpositive, fatherId=fReference[0]}
  [446] = {x=-372, y=-44, z=132, rx=-180, rz=85.171, shoulder=lefty, elbow=epositive, wrist=wpositive, fatherId=fReference[0]}
  [447] = {x=-369.477, y=-73.864, z=132, rx=-180, rz=75.512, shoulder=lefty, elbow=epositive, wrist=wpositive, fatherId=fReference[0]}
  [448] = {x=-361.979, y=-102.881, z=132, rx=-180, rz=65.854, shoulder=lefty, elbow=epositive, wrist=wpositive, fatherId=fReference[0]}
  [449] = {x=-349.719, y=-130.229, z=132, rx=-180, rz=56.195, shoulder=lefty, elbow=epositive, wrist=wpositive, fatherId=fReference[0]}
  [450] = {x=-333.045, y=-155.133, z=132, rx=-180, rz=46.537, shoulder=lefty, elbow=epositive, wrist=wpositive, fatherId=fReference[0]}
  [451] = {x=-312.429, y=-176.886, z=132, rx=-180, rz=36.878, shoulder=lefty, elbow=epositive, wrist=wpositive, fatherId=fReference[0]}
  [452] = {x=-288.455, y=-194.872, z=132, rx=-180, rz=27.22, shoulder=lefty, elbow=epositive, wrist=wpositive, fatherId=fReference[0]}
  [453] = {x=-261.803, y=-208.58, z=132, rx=180, rz=17.561, shoulder=lefty, elbow=epositive, wrist=wpositive, fatherId=fReference[0]}
  [454] = {x=-233.23, y=-217.623, z=132, rx=180, rz=7.903, shoulder=lefty, elbow=epositive, wrist=wpositive, fatherId=fReference[0]}
  [455] = {x=-203.544, y=-221.744, z=132, rx=-180, rz=0.489, shoulder=lefty, elbow=epositive, wrist=wpositive, fatherId=fReference[0]}
  [456] = {x=-173.543, y=-222, z=132, rx=180, shoulder=lefty, elbow=epositive, wrist=wpositive, fatherId=fReference[0]}
  [457] = {x=-143.537, y=-222, z=132, rx=-180, shoulder=lefty, elbow=epositive, wrist=wpositive, fatherId=fReference[0]}
  [458] = {x=-113.531, y=-222, z=132, rx=-180, shoulder=lefty, elbow=epositive, wrist=wpositive, fatherId=fReference[0]}
  [459] = {x=-83.525, y=-222, z=132, rx=180, shoulder=lefty, elbow=epositive, wrist=wpositive, fatherId=fReference[0]}
  [460] = {x=-53.519, y=-222, z=132, rx=180, shoulder=lefty, elbow=epositive, wrist=wpositive, fatherId=fReference[0]}
  [461] = {x=-23.513, y=-222, z=132, rx=180, shoulder=lefty, elbow=epositive, wrist=wpositive, fatherId=fReference[0]}
  [462] = {x=6.493, y=-222, z=132, rx=-180, shoulder=lefty, elbow=epositive, wrist=wpositive, fatherId=fReference[0]}
  [463] = {x=36.499, y=-222, z=132, rx=-180, shoulder=lefty, elbow=epositive, wrist=wpositive, fatherId=fReference[0]}
  [464] = {x=66.504, y=-222, z=132, rx=-180, shoulder=lefty, elbow=epositive, wrist=wpositive, fatherId=fReference[0]}
  [465] = {x=96.51, y=-222, z=132, rx=-180, shoulder=lefty, elbow=epositive, wrist=wpositive, fatherId=fReference[0]}
  [466] = {x=126.516, y=-222, z=132, rx=180, shoulder=lefty, elbow=epositive, wrist=wpositive, fatherId=fReference[0]}
  [467] = {x=156.522, y=-222, z=132, rx=-180, shoulder=lefty, elbow=epositive, wrist=wpositive, fatherId=fReference[0]}
  [468] = {x=186.528, y=-222, z=132, rx=180, rz=-2.723, shoulder=lefty, elbow=epositive, wrist=wpositive, fatherId=fReference[0]}
  [469] = {x=216.474, y=-220.576, z=132, rx=-180, rz=-12.083, shoulder=lefty, elbow=epositive, wrist=wpositive, fatherId=fReference[0]}
  [470] = {x=245.78, y=-214.302, z=132, rx=180, rz=-21.741, shoulder=lefty, elbow=epositive, wrist=wpositive, fatherId=fReference[0]}
  [471] = {x=273.619, y=-203.201, z=132, rx=-180, rz=-31.4, shoulder=lefty, elbow=epositive, wrist=wpositive, fatherId=fReference[0]}
  [472] = {x=299.2, y=-187.586, z=132, rx=-180, rz=-41.058, shoulder=lefty, elbow=epositive, wrist=wpositive, fatherId=fReference[0]}
  [473] = {x=321.799, y=-167.901, z=132, rx=-180, rz=-50.717, shoulder=lefty, elbow=epositive, wrist=wpositive, fatherId=fReference[0]}
  [474] = {x=340.775, y=-144.703, z=132, rx=-180, rz=-60.375, shoulder=lefty, elbow=epositive, wrist=wpositive, fatherId=fReference[0]}
  [475] = {x=355.59, y=-118.65, z=132, rx=180, rz=-70.034, shoulder=lefty, elbow=epositive, wrist=wpositive, fatherId=fReference[0]}
  [476] = {x=365.824, y=-90.481, z=132, rx=180, rz=-79.692, shoulder=lefty, elbow=epositive, wrist=wpositive, fatherId=fReference[0]}
  [477] = {x=371.187, y=-60.995, z=132, rx=180, rz=-88.446, shoulder=lefty, elbow=epositive, wrist=wpositive, fatherId=fReference[0]}
  [478] = {x=372, y=-31.015, z=132, rx=180, rz=-90, shoulder=lefty, elbow=epositive, wrist=wpositive, fatherId=fReference[0]}
  [479] = {x=372, y=-1.009, z=132, rx=180, rz=-90, shoulder=lefty, elbow=epositive, wrist=wpositive, fatherId=fReference[0]}
  [480] = {x=372, y=28.997, z=132, rx=-180, rz=-91.207, shoulder=lefty, elbow=epositive, wrist=wpositive, fatherId=fReference[0]}
  [481] = {x=371.368, y=58.985, z=132, rx=-180, rz=-99.658, shoulder=lefty, elbow=epositive, wrist=wpositive, fatherId=fReference[0]}
  [482] = {x=366.34, y=88.531, z=132, rx=-180, rz=-109.317, shoulder=lefty, elbow=epositive, wrist=wpositive, fatherId=fReference[0]}
  [483] = {x=356.426, y=116.814, z=132, rx=-180, rz=-118.975, shoulder=lefty, elbow=epositive, wrist=wpositive, fatherId=fReference[0]}
  [484] = {x=341.907, y=143.033, z=132, rx=-180, rz=-128.634, shoulder=lefty, elbow=epositive, wrist=wpositive, fatherId=fReference[0]}
  [485] = {x=323.195, y=166.444, z=132, rx=-180, rz=-138.292, shoulder=lefty, elbow=epositive, wrist=wpositive, fatherId=fReference[0]}
  [486] = {x=300.821, y=186.384, z=132, rx=-180, rz=-147.951, shoulder=lefty, elbow=epositive, wrist=wpositive, fatherId=fReference[0]}
  [487] = {x=275.418, y=202.288, z=132, rx=180, rz=-157.609, shoulder=lefty, elbow=epositive, wrist=wpositive, fatherId=fReference[0]}
  [488] = {x=247.707, y=213.704, z=132, rx=-180, rz=-167.268, shoulder=lefty, elbow=epositive, wrist=wpositive, fatherId=fReference[0]}
  [489] = {x=218.474, y=220.309, z=132, rx=-180, rz=-176.767, shoulder=lefty, elbow=epositive, wrist=wpositive, fatherId=fReference[0]}
  [490] = {x=188.546, y=222, z=132, rx=-180, rz=180, shoulder=lefty, elbow=epositive, wrist=wpositive, fatherId=fReference[0]}
  [491] = {x=158.54, y=222, z=132, rx=180, rz=-180, shoulder=lefty, elbow=epositive, wrist=wpositive, fatherId=fReference[0]}
  [492] = {x=128.534, y=222, z=132, rx=180, rz=-180, shoulder=lefty, elbow=epositive, wrist=wpositive, fatherId=fReference[0]}
  [493] = {x=98.528, y=222, z=132, rx=-180, rz=-180, shoulder=lefty, elbow=epositive, wrist=wpositive, fatherId=fReference[0]}
  [494] = {x=68.522, y=222, z=132, rx=-180, rz=-180, shoulder=lefty, elbow=epositive, wrist=wpositive, fatherId=fReference[0]}
  [495] = {x=38.516, y=222, z=132, rx=180, rz=-180, shoulder=lefty, elbow=epositive, wrist=wpositive, fatherId=fReference[0]}
  [496] = {x=8.51, y=222, z=132, rx=180, rz=-180, shoulder=lefty, elbow=epositive, wrist=wpositive, fatherId=fReference[0]}
  [497] = {x=-21.496, y=222, z=132, rx=-180, rz=-180, shoulder=lefty, elbow=epositive, wrist=wpositive, fatherId=fReference[0]}
  [498] = {x=-51.501, y=222, z=132, rx=180, rz=-180, shoulder=lefty, elbow=epositive, wrist=wpositive, fatherId=fReference[0]}
  [499] = {x=-81.507, y=222, z=132, rx=-180, rz=-180, shoulder=lefty, elbow=epositive, wrist=wpositive, fatherId=fReference[0]}
  [500] = {x=-111.513, y=222, z=132, rx=180, rz=-180, shoulder=lefty, elbow=epositive, wrist=wpositive, fatherId=fReference[0]}
  [501] = {x=-141.519, y=222, z=132, rx=180, rz=-180, shoulder=lefty, elbow=epositive, wrist=wpositive, fatherId=fReference[0]}
  [502] = {x=-171.525, y=222, z=132, rx=180, rz=179.696, shoulder=lefty, elbow=epositive, wrist=wpositive, fatherId=fReference[0]}
  [503] = {x=-201.529, y=221.841, z=132, rx=180, rz=172.747, shoulder=lefty, elbow=epositive, wrist=wpositive, fatherId=fReference[0]}
  [504] = {x=-231.259, y=218.057, z=132, rx=-180, rz=163.088, shoulder=lefty, elbow=epositive, wrist=wpositive, fatherId=fReference[0]}
  [505] = {x=-259.934, y=209.338, z=132, rx=180, rz=153.43, shoulder=lefty, elbow=epositive, wrist=wpositive, fatherId=fReference[0]}
  [506] = {x=-286.739, y=195.933, z=132, rx=180, rz=143.771, shoulder=lefty, elbow=epositive, wrist=wpositive, fatherId=fReference[0]}
  [507] = {x=-310.915, y=178.22, z=132, rx=180, rz=134.113, shoulder=lefty, elbow=epositive, wrist=wpositive, fatherId=fReference[0]}
  [508] = {x=-331.776, y=156.702, z=132, rx=180, rz=124.454, shoulder=lefty, elbow=epositive, wrist=wpositive, fatherId=fReference[0]}
  [509] = {x=-348.732, y=131.989, z=132, rx=180, rz=114.796, shoulder=lefty, elbow=epositive, wrist=wpositive, fatherId=fReference[0]}
  [510] = {x=-361.301, y=104.782, z=132, rx=180, rz=105.137, shoulder=lefty, elbow=epositive, wrist=wpositive, fatherId=fReference[0]}
  [511] = {x=-369.127, y=75.851, z=132, rx=180, rz=95.479, shoulder=lefty, elbow=epositive, wrist=wpositive, fatherId=fReference[0]}
  [512] = {x=-371.989, y=46.018, z=132, rx=180, rz=90.022, shoulder=lefty, elbow=epositive, wrist=wpositive, fatherId=fReference[0]}
  [513] = {x=-372, y=16.012, z=132, rx=-180, rz=90, shoulder=lefty, elbow=epositive, wrist=wpositive, fatherId=fReference[0]}
  [514] = {x=-372, y=-13.994, z=132, rx=-180, rz=90, shoulder=lefty, elbow=epositive, wrist=wpositive, fatherId=fReference[0]}
  [515] = {x=-372, y=-44, z=132, rx=-180, rz=90, shoulder=lefty, elbow=epositive, wrist=wpositive, fatherId=fReference[0]}
  [516] = {x=-372, y=-44, z=132, rx=-180, rz=90, shoulder=lefty, elbow=epositive, wrist=wpositive, fatherId=fReference[0]}
  [517] = {x=-372, y=-44, z=232, rx=-180, rz=90, shoulder=lefty, elbow=epositive, wrist=wpositive, fatherId=fReference[0]}
  [518] = {x=-372, y=-44, z=254, rx=-180, rz=90, shoulder=lefty, elbow=epositive, wrist=wpositive, fatherId=fReference[0]}
  [519] = {x=-372, y=-44, z=154, rx=-180, rz=90, shoulder=lefty, elbow=epositive, wrist=wpositive, fatherId=fReference[0]}
  [520] = {x=-372, y=-44, z=154, rx=-180, rz=90, shoulder=lefty, elbow=epositive, wrist=wpositive, fatherId=fReference[0]}
  [521] = {x=-372, y=-13.994, z=154, rx=-180, rz=90, shoulder=lefty, elbow=epositive, wrist=wpositive, fatherId=fReference[0]}
  [522] = {x=-372, y=16.012, z=154, rx=180, rz=90.022, shoulder=lefty, elbow=epositive, wrist=wpositive, fatherId=fReference[0]}
  [523] = {x=-371.989, y=46.018, z=154, rx=180, rz=95.479, shoulder=lefty, elbow=epositive, wrist=wpositive, fatherId=fReference[0]}
  [524] = {x=-369.127, y=75.851, z=154, rx=180, rz=105.137, shoulder=lefty, elbow=epositive, wrist=wpositive, fatherId=fReference[0]}
  [525] = {x=-361.301, y=104.782, z=154, rx=180, rz=114.796, shoulder=lefty, elbow=epositive, wrist=wpositive, fatherId=fReference[0]}
  [526] = {x=-348.732, y=131.989, z=154, rx=180, rz=124.454, shoulder=lefty, elbow=epositive, wrist=wpositive, fatherId=fReference[0]}
  [527] = {x=-331.776, y=156.702, z=154, rx=-180, rz=134.113, shoulder=lefty, elbow=epositive, wrist=wpositive, fatherId=fReference[0]}
  [528] = {x=-310.915, y=178.22, z=154, rx=180, rz=143.771, shoulder=lefty, elbow=epositive, wrist=wpositive, fatherId=fReference[0]}
  [529] = {x=-286.739, y=195.933, z=154, rx=180, rz=153.43, shoulder=lefty, elbow=epositive, wrist=wpositive, fatherId=fReference[0]}
  [530] = {x=-259.934, y=209.338, z=154, rx=180, rz=163.088, shoulder=lefty, elbow=epositive, wrist=wpositive, fatherId=fReference[0]}
  [531] = {x=-231.259, y=218.057, z=154, rx=-180, rz=172.747, shoulder=lefty, elbow=epositive, wrist=wpositive, fatherId=fReference[0]}
  [532] = {x=-201.529, y=221.841, z=154, rx=180, rz=179.696, shoulder=lefty, elbow=epositive, wrist=wpositive, fatherId=fReference[0]}
  [533] = {x=-171.525, y=222, z=154, rx=-180, rz=180, shoulder=lefty, elbow=epositive, wrist=wpositive, fatherId=fReference[0]}
  [534] = {x=-141.519, y=222, z=154, rx=180, rz=-180, shoulder=lefty, elbow=epositive, wrist=wpositive, fatherId=fReference[0]}
  [535] = {x=-111.513, y=222, z=154, rx=-180, rz=-180, shoulder=lefty, elbow=epositive, wrist=wpositive, fatherId=fReference[0]}
  [536] = {x=-81.507, y=222, z=154, rx=180, rz=-180, shoulder=lefty, elbow=epositive, wrist=wpositive, fatherId=fReference[0]}
  [537] = {x=-51.501, y=222, z=154, rx=180, rz=-180, shoulder=lefty, elbow=epositive, wrist=wpositive, fatherId=fReference[0]}
  [538] = {x=-21.496, y=222, z=154, rx=-180, rz=-180, shoulder=lefty, elbow=epositive, wrist=wpositive, fatherId=fReference[0]}
  [539] = {x=8.51, y=222, z=154, rx=180, rz=-180, shoulder=lefty, elbow=epositive, wrist=wpositive, fatherId=fReference[0]}
  [540] = {x=38.516, y=222, z=154, rx=-180, rz=-180, shoulder=lefty, elbow=epositive, wrist=wpositive, fatherId=fReference[0]}
  [541] = {x=68.522, y=222, z=154, rx=180, rz=-180, shoulder=lefty, elbow=epositive, wrist=wpositive, fatherId=fReference[0]}
  [542] = {x=98.528, y=222, z=154, rx=-180, rz=-180, shoulder=lefty, elbow=epositive, wrist=wpositive, fatherId=fReference[0]}
  [543] = {x=128.534, y=222, z=154, rx=-180, rz=-180, shoulder=lefty, elbow=epositive, wrist=wpositive, fatherId=fReference[0]}
  [544] = {x=158.54, y=222, z=154, rx=-180, rz=-180, shoulder=lefty, elbow=epositive, wrist=wpositive, fatherId=fReference[0]}
  [545] = {x=188.546, y=222, z=154, rx=-180, rz=-176.767, shoulder=lefty, elbow=epositive, wrist=wpositive, fatherId=fReference[0]}
  [546] = {x=218.474, y=220.309, z=154, rx=-180, rz=-167.268, shoulder=lefty, elbow=epositive, wrist=wpositive, fatherId=fReference[0]}
  [547] = {x=247.707, y=213.704, z=154, rx=-180, rz=-157.609, shoulder=lefty, elbow=epositive, wrist=wpositive, fatherId=fReference[0]}
  [548] = {x=275.418, y=202.288, z=154, rx=-180, rz=-147.951, shoulder=lefty, elbow=epositive, wrist=wpositive, fatherId=fReference[0]}
  [549] = {x=300.821, y=186.384, z=154, rx=-180, rz=-138.292, shoulder=lefty, elbow=epositive, wrist=wpositive, fatherId=fReference[0]}
  [550] = {x=323.195, y=166.444, z=154, rx=-180, rz=-128.634, shoulder=lefty, elbow=epositive, wrist=wpositive, fatherId=fReference[0]}
  [551] = {x=341.907, y=143.033, z=154, rx=-180, rz=-118.975, shoulder=lefty, elbow=epositive, wrist=wpositive, fatherId=fReference[0]}
  [552] = {x=356.426, y=116.814, z=154, rx=-180, rz=-109.317, shoulder=lefty, elbow=epositive, wrist=wpositive, fatherId=fReference[0]}
  [553] = {x=366.34, y=88.531, z=154, rx=-180, rz=-99.658, shoulder=lefty, elbow=epositive, wrist=wpositive, fatherId=fReference[0]}
  [554] = {x=371.368, y=58.985, z=154, rx=-180, rz=-91.207, shoulder=lefty, elbow=epositive, wrist=wpositive, fatherId=fReference[0]}
  [555] = {x=372, y=28.997, z=154, rx=180, rz=-90, shoulder=lefty, elbow=epositive, wrist=wpositive, fatherId=fReference[0]}
  [556] = {x=372, y=-1.009, z=154, rx=180, rz=-90, shoulder=lefty, elbow=epositive, wrist=wpositive, fatherId=fReference[0]}
  [557] = {x=372, y=-31.015, z=154, rx=180, rz=-88.446, shoulder=lefty, elbow=epositive, wrist=wpositive, fatherId=fReference[0]}
  [558] = {x=371.187, y=-60.995, z=154, rx=180, rz=-79.692, shoulder=lefty, elbow=epositive, wrist=wpositive, fatherId=fReference[0]}
  [559] = {x=365.824, y=-90.481, z=154, rx=180, rz=-70.034, shoulder=lefty, elbow=epositive, wrist=wpositive, fatherId=fReference[0]}
  [560] = {x=355.59, y=-118.65, z=154, rx=180, rz=-60.375, shoulder=lefty, elbow=epositive, wrist=wpositive, fatherId=fReference[0]}
  [561] = {x=340.775, y=-144.703, z=154, rx=180, rz=-50.717, shoulder=lefty, elbow=epositive, wrist=wpositive, fatherId=fReference[0]}
  [562] = {x=321.799, y=-167.901, z=154, rx=180, rz=-41.058, shoulder=lefty, elbow=epositive, wrist=wpositive, fatherId=fReference[0]}
  [563] = {x=299.2, y=-187.586, z=154, rx=180, rz=-31.4, shoulder=lefty, elbow=epositive, wrist=wpositive, fatherId=fReference[0]}
  [564] = {x=273.619, y=-203.201, z=154, rx=180, rz=-21.741, shoulder=lefty, elbow=epositive, wrist=wpositive, fatherId=fReference[0]}
  [565] = {x=245.78, y=-214.302, z=154, rx=180, rz=-12.083, shoulder=lefty, elbow=epositive, wrist=wpositive, fatherId=fReference[0]}
  [566] = {x=216.474, y=-220.576, z=154, rx=180, rz=-2.723, shoulder=lefty, elbow=epositive, wrist=wpositive, fatherId=fReference[0]}
  [567] = {x=186.528, y=-222, z=154, rx=180, shoulder=lefty, elbow=epositive, wrist=wpositive, fatherId=fReference[0]}
  [568] = {x=156.522, y=-222, z=154, rx=-180, shoulder=lefty, elbow=epositive, wrist=wpositive, fatherId=fReference[0]}
  [569] = {x=126.516, y=-222, z=154, rx=-180, shoulder=lefty, elbow=epositive, wrist=wpositive, fatherId=fReference[0]}
  [570] = {x=96.51, y=-222, z=154, rx=180, shoulder=lefty, elbow=epositive, wrist=wpositive, fatherId=fReference[0]}
  [571] = {x=66.504, y=-222, z=154, rx=-180, shoulder=lefty, elbow=epositive, wrist=wpositive, fatherId=fReference[0]}
  [572] = {x=36.499, y=-222, z=154, rx=-180, shoulder=lefty, elbow=epositive, wrist=wpositive, fatherId=fReference[0]}
  [573] = {x=6.493, y=-222, z=154, rx=-180, shoulder=lefty, elbow=epositive, wrist=wpositive, fatherId=fReference[0]}
  [574] = {x=-23.513, y=-222, z=154, rx=180, shoulder=lefty, elbow=epositive, wrist=wpositive, fatherId=fReference[0]}
  [575] = {x=-53.519, y=-222, z=154, rx=-180, shoulder=lefty, elbow=epositive, wrist=wpositive, fatherId=fReference[0]}
  [576] = {x=-83.525, y=-222, z=154, rx=180, shoulder=lefty, elbow=epositive, wrist=wpositive, fatherId=fReference[0]}
  [577] = {x=-113.531, y=-222, z=154, rx=-180, shoulder=lefty, elbow=epositive, wrist=wpositive, fatherId=fReference[0]}
  [578] = {x=-143.537, y=-222, z=154, rx=180, shoulder=lefty, elbow=epositive, wrist=wpositive, fatherId=fReference[0]}
  [579] = {x=-173.543, y=-222, z=154, rx=180, rz=0.489, shoulder=lefty, elbow=epositive, wrist=wpositive, fatherId=fReference[0]}
  [580] = {x=-203.544, y=-221.744, z=154, rx=-180, rz=7.903, shoulder=lefty, elbow=epositive, wrist=wpositive, fatherId=fReference[0]}
  [581] = {x=-233.23, y=-217.623, z=154, rx=-180, rz=17.561, shoulder=lefty, elbow=epositive, wrist=wpositive, fatherId=fReference[0]}
  [582] = {x=-261.803, y=-208.58, z=154, rx=180, rz=27.22, shoulder=lefty, elbow=epositive, wrist=wpositive, fatherId=fReference[0]}
  [583] = {x=-288.455, y=-194.872, z=154, rx=-180, rz=36.878, shoulder=lefty, elbow=epositive, wrist=wpositive, fatherId=fReference[0]}
  [584] = {x=-312.429, y=-176.886, z=154, rx=-180, rz=46.537, shoulder=lefty, elbow=epositive, wrist=wpositive, fatherId=fReference[0]}
  [585] = {x=-333.045, y=-155.133, z=154, rx=-180, rz=56.195, shoulder=lefty, elbow=epositive, wrist=wpositive, fatherId=fReference[0]}
  [586] = {x=-349.719, y=-130.229, z=154, rx=-180, rz=65.854, shoulder=lefty, elbow=epositive, wrist=wpositive, fatherId=fReference[0]}
  [587] = {x=-361.979, y=-102.881, z=154, rx=-180, rz=75.512, shoulder=lefty, elbow=epositive, wrist=wpositive, fatherId=fReference[0]}
  [588] = {x=-369.477, y=-73.864, z=154, rx=-180, rz=85.171, shoulder=lefty, elbow=epositive, wrist=wpositive, fatherId=fReference[0]}
  [589] = {x=-372, y=-44, z=154, rx=-180, rz=85.171, shoulder=lefty, elbow=epositive, wrist=wpositive, fatherId=fReference[0]}
  [590] = {x=-372, y=-44, z=154, rx=-180, rz=85.171, shoulder=lefty, elbow=epositive, wrist=wpositive, fatherId=fReference[0]}
  [591] = {x=-372, y=-44, z=254, rx=-180, rz=85.171, shoulder=lefty, elbow=epositive, wrist=wpositive, fatherId=fReference[0]}
  [592] = {x=-372, y=-44, z=276, rx=-180, rz=85.171, shoulder=lefty, elbow=epositive, wrist=wpositive, fatherId=fReference[0]}
  [593] = {x=-372, y=-44, z=176, rx=-180, rz=85.171, shoulder=lefty, elbow=epositive, wrist=wpositive, fatherId=fReference[0]}
  [594] = {x=-372, y=-44, z=176, rx=-180, rz=85.171, shoulder=lefty, elbow=epositive, wrist=wpositive, fatherId=fReference[0]}
  [595] = {x=-369.477, y=-73.864, z=176, rx=-180, rz=75.512, shoulder=lefty, elbow=epositive, wrist=wpositive, fatherId=fReference[0]}
  [596] = {x=-361.979, y=-102.881, z=176, rx=-180, rz=65.854, shoulder=lefty, elbow=epositive, wrist=wpositive, fatherId=fReference[0]}
  [597] = {x=-349.719, y=-130.229, z=176, rx=180, rz=56.195, shoulder=lefty, elbow=epositive, wrist=wpositive, fatherId=fReference[0]}
  [598] = {x=-333.045, y=-155.133, z=176, rx=-180, rz=46.537, shoulder=lefty, elbow=epositive, wrist=wpositive, fatherId=fReference[0]}
  [599] = {x=-312.429, y=-176.886, z=176, rx=180, rz=36.878, shoulder=lefty, elbow=epositive, wrist=wpositive, fatherId=fReference[0]}
  [600] = {x=-288.455, y=-194.872, z=176, rx=-180, rz=27.22, shoulder=lefty, elbow=epositive, wrist=wpositive, fatherId=fReference[0]}
  [601] = {x=-261.803, y=-208.58, z=176, rx=-180, rz=17.561, shoulder=lefty, elbow=epositive, wrist=wpositive, fatherId=fReference[0]}
  [602] = {x=-233.23, y=-217.623, z=176, rx=-180, rz=7.903, shoulder=lefty, elbow=epositive, wrist=wpositive, fatherId=fReference[0]}
  [603] = {x=-203.544, y=-221.744, z=176, rx=180, rz=0.489, shoulder=lefty, elbow=epositive, wrist=wpositive, fatherId=fReference[0]}
  [604] = {x=-173.543, y=-222, z=176, rx=-180, shoulder=lefty, elbow=epositive, wrist=wpositive, fatherId=fReference[0]}
  [605] = {x=-143.537, y=-222, z=176, rx=180, shoulder=lefty, elbow=epositive, wrist=wpositive, fatherId=fReference[0]}
  [606] = {x=-113.531, y=-222, z=176, rx=-180, shoulder=lefty, elbow=epositive, wrist=wpositive, fatherId=fReference[0]}
  [607] = {x=-83.525, y=-222, z=176, rx=180, shoulder=lefty, elbow=epositive, wrist=wpositive, fatherId=fReference[0]}
  [608] = {x=-53.519, y=-222, z=176, rx=180, shoulder=lefty, elbow=epositive, wrist=wpositive, fatherId=fReference[0]}
  [609] = {x=-23.513, y=-222, z=176, rx=-180, shoulder=lefty, elbow=epositive, wrist=wpositive, fatherId=fReference[0]}
  [610] = {x=6.493, y=-222, z=176, rx=-180, shoulder=lefty, elbow=epositive, wrist=wpositive, fatherId=fReference[0]}
  [611] = {x=36.499, y=-222, z=176, rx=-180, shoulder=lefty, elbow=epositive, wrist=wpositive, fatherId=fReference[0]}
  [612] = {x=66.504, y=-222, z=176, rx=-180, shoulder=lefty, elbow=epositive, wrist=wpositive, fatherId=fReference[0]}
  [613] = {x=96.51, y=-222, z=176, rx=-180, shoulder=lefty, elbow=epositive, wrist=wpositive, fatherId=fReference[0]}
  [614] = {x=126.516, y=-222, z=176, rx=180, shoulder=lefty, elbow=epositive, wrist=wpositive, fatherId=fReference[0]}
  [615] = {x=156.522, y=-222, z=176, rx=-180, shoulder=lefty, elbow=epositive, wrist=wpositive, fatherId=fReference[0]}
  [616] = {x=186.528, y=-222, z=176, rx=180, rz=-2.723, shoulder=lefty, elbow=epositive, wrist=wpositive, fatherId=fReference[0]}
  [617] = {x=216.474, y=-220.576, z=176, rx=180, rz=-12.083, shoulder=lefty, elbow=epositive, wrist=wpositive, fatherId=fReference[0]}
  [618] = {x=245.78, y=-214.302, z=176, rx=-180, rz=-21.741, shoulder=lefty, elbow=epositive, wrist=wpositive, fatherId=fReference[0]}
  [619] = {x=273.619, y=-203.201, z=176, rx=-180, rz=-31.4, shoulder=lefty, elbow=epositive, wrist=wpositive, fatherId=fReference[0]}
  [620] = {x=299.2, y=-187.586, z=176, rx=-180, rz=-41.058, shoulder=lefty, elbow=epositive, wrist=wpositive, fatherId=fReference[0]}
  [621] = {x=321.799, y=-167.901, z=176, rx=-180, rz=-50.717, shoulder=lefty, elbow=epositive, wrist=wpositive, fatherId=fReference[0]}
  [622] = {x=340.775, y=-144.703, z=176, rx=180, rz=-60.375, shoulder=lefty, elbow=epositive, wrist=wpositive, fatherId=fReference[0]}
  [623] = {x=355.59, y=-118.65, z=176, rx=-180, rz=-70.034, shoulder=lefty, elbow=epositive, wrist=wpositive, fatherId=fReference[0]}
  [624] = {x=365.824, y=-90.481, z=176, rx=180, rz=-79.692, shoulder=lefty, elbow=epositive, wrist=wpositive, fatherId=fReference[0]}
  [625] = {x=371.187, y=-60.995, z=176, rx=180, rz=-88.446, shoulder=lefty, elbow=epositive, wrist=wpositive, fatherId=fReference[0]}
  [626] = {x=372, y=-31.015, z=176, rx=180, rz=-90, shoulder=lefty, elbow=epositive, wrist=wpositive, fatherId=fReference[0]}
  [627] = {x=372, y=-1.009, z=176, rx=180, rz=-90, shoulder=lefty, elbow=epositive, wrist=wpositive, fatherId=fReference[0]}
  [628] = {x=372, y=28.997, z=176, rx=-180, rz=-91.207, shoulder=lefty, elbow=epositive, wrist=wpositive, fatherId=fReference[0]}
  [629] = {x=371.368, y=58.985, z=176, rx=-180, rz=-99.658, shoulder=lefty, elbow=epositive, wrist=wpositive, fatherId=fReference[0]}
  [630] = {x=366.34, y=88.531, z=176, rx=-180, rz=-109.317, shoulder=lefty, elbow=epositive, wrist=wpositive, fatherId=fReference[0]}
  [631] = {x=356.426, y=116.814, z=176, rx=-180, rz=-118.975, shoulder=lefty, elbow=epositive, wrist=wpositive, fatherId=fReference[0]}
  [632] = {x=341.907, y=143.033, z=176, rx=-180, rz=-128.634, shoulder=lefty, elbow=epositive, wrist=wpositive, fatherId=fReference[0]}
  [633] = {x=323.195, y=166.444, z=176, rx=-180, rz=-138.292, shoulder=lefty, elbow=epositive, wrist=wpositive, fatherId=fReference[0]}
  [634] = {x=300.821, y=186.384, z=176, rx=-180, rz=-147.951, shoulder=lefty, elbow=epositive, wrist=wpositive, fatherId=fReference[0]}
  [635] = {x=275.418, y=202.288, z=176, rx=-180, rz=-157.609, shoulder=lefty, elbow=epositive, wrist=wpositive, fatherId=fReference[0]}
  [636] = {x=247.707, y=213.704, z=176, rx=-180, rz=-167.268, shoulder=lefty, elbow=epositive, wrist=wpositive, fatherId=fReference[0]}
  [637] = {x=218.474, y=220.309, z=176, rx=180, rz=-176.767, shoulder=lefty, elbow=epositive, wrist=wpositive, fatherId=fReference[0]}
  [638] = {x=188.546, y=222, z=176, rx=180, rz=-180, shoulder=lefty, elbow=epositive, wrist=wpositive, fatherId=fReference[0]}
  [639] = {x=158.54, y=222, z=176, rx=180, rz=-180, shoulder=lefty, elbow=epositive, wrist=wpositive, fatherId=fReference[0]}
  [640] = {x=128.534, y=222, z=176, rx=180, rz=-180, shoulder=lefty, elbow=epositive, wrist=wpositive, fatherId=fReference[0]}
  [641] = {x=98.528, y=222, z=176, rx=-180, rz=-180, shoulder=lefty, elbow=epositive, wrist=wpositive, fatherId=fReference[0]}
  [642] = {x=68.522, y=222, z=176, rx=180, rz=-180, shoulder=lefty, elbow=epositive, wrist=wpositive, fatherId=fReference[0]}
  [643] = {x=38.516, y=222, z=176, rx=-180, rz=-180, shoulder=lefty, elbow=epositive, wrist=wpositive, fatherId=fReference[0]}
  [644] = {x=8.51, y=222, z=176, rx=-180, rz=-180, shoulder=lefty, elbow=epositive, wrist=wpositive, fatherId=fReference[0]}
  [645] = {x=-21.496, y=222, z=176, rx=180, rz=-180, shoulder=lefty, elbow=epositive, wrist=wpositive, fatherId=fReference[0]}
  [646] = {x=-51.501, y=222, z=176, rx=-180, rz=-180, shoulder=lefty, elbow=epositive, wrist=wpositive, fatherId=fReference[0]}
  [647] = {x=-81.507, y=222, z=176, rx=-180, rz=-180, shoulder=lefty, elbow=epositive, wrist=wpositive, fatherId=fReference[0]}
  [648] = {x=-111.513, y=222, z=176, rx=-180, rz=-180, shoulder=lefty, elbow=epositive, wrist=wpositive, fatherId=fReference[0]}
  [649] = {x=-141.519, y=222, z=176, rx=-180, rz=-180, shoulder=lefty, elbow=epositive, wrist=wpositive, fatherId=fReference[0]}
  [650] = {x=-171.525, y=222, z=176, rx=-180, rz=179.696, shoulder=lefty, elbow=epositive, wrist=wpositive, fatherId=fReference[0]}
  [651] = {x=-201.529, y=221.841, z=176, rx=-180, rz=172.747, shoulder=lefty, elbow=epositive, wrist=wpositive, fatherId=fReference[0]}
  [652] = {x=-231.259, y=218.057, z=176, rx=180, rz=163.088, shoulder=lefty, elbow=epositive, wrist=wpositive, fatherId=fReference[0]}
  [653] = {x=-259.934, y=209.338, z=176, rx=180, rz=153.43, shoulder=lefty, elbow=epositive, wrist=wpositive, fatherId=fReference[0]}
  [654] = {x=-286.739, y=195.933, z=176, rx=180, rz=143.771, shoulder=lefty, elbow=epositive, wrist=wpositive, fatherId=fReference[0]}
  [655] = {x=-310.915, y=178.22, z=176, rx=180, rz=134.113, shoulder=lefty, elbow=epositive, wrist=wpositive, fatherId=fReference[0]}
  [656] = {x=-331.776, y=156.702, z=176, rx=180, rz=124.454, shoulder=lefty, elbow=epositive, wrist=wpositive, fatherId=fReference[0]}
  [657] = {x=-348.732, y=131.989, z=176, rx=180, rz=114.796, shoulder=lefty, elbow=epositive, wrist=wpositive, fatherId=fReference[0]}
  [658] = {x=-361.301, y=104.782, z=176, rx=180, rz=105.137, shoulder=lefty, elbow=epositive, wrist=wpositive, fatherId=fReference[0]}
  [659] = {x=-369.127, y=75.851, z=176, rx=180, rz=95.479, shoulder=lefty, elbow=epositive, wrist=wpositive, fatherId=fReference[0]}
  [660] = {x=-371.989, y=46.018, z=176, rx=180, rz=90.022, shoulder=lefty, elbow=epositive, wrist=wpositive, fatherId=fReference[0]}
  [661] = {x=-372, y=16.012, z=176, rx=180, rz=90, shoulder=lefty, elbow=epositive, wrist=wpositive, fatherId=fReference[0]}
  [662] = {x=-372, y=-13.994, z=176, rx=180, rz=90, shoulder=lefty, elbow=epositive, wrist=wpositive, fatherId=fReference[0]}
  [663] = {x=-372, y=-44, z=176, rx=180, rz=90, shoulder=lefty, elbow=epositive, wrist=wpositive, fatherId=fReference[0]}
  [664] = {x=-372, y=-44, z=176, rx=180, rz=90, shoulder=lefty, elbow=epositive, wrist=wpositive, fatherId=fReference[0]}
  [665] = {x=-372, y=-44, z=276, rx=180, rz=90, shoulder=lefty, elbow=epositive, wrist=wpositive, fatherId=fReference[0]}
  [666] = {x=-372, y=-44, z=298, rx=180, rz=90, shoulder=lefty, elbow=epositive, wrist=wpositive, fatherId=fReference[0]}
  [667] = {x=-372, y=-44, z=198, rx=180, rz=90, shoulder=lefty, elbow=epositive, wrist=wpositive, fatherId=fReference[0]}
  [668] = {x=-372, y=-44, z=198, rx=180, rz=90, shoulder=lefty, elbow=epositive, wrist=wpositive, fatherId=fReference[0]}
  [669] = {x=-372, y=-13.994, z=198, rx=180, rz=90, shoulder=lefty, elbow=epositive, wrist=wpositive, fatherId=fReference[0]}
  [670] = {x=-372, y=16.012, z=198, rx=180, rz=90.022, shoulder=lefty, elbow=epositive, wrist=wpositive, fatherId=fReference[0]}
  [671] = {x=-371.989, y=46.018, z=198, rx=180, rz=95.479, shoulder=lefty, elbow=epositive, wrist=wpositive, fatherId=fReference[0]}
  [672] = {x=-369.127, y=75.851, z=198, rx=180, rz=105.137, shoulder=lefty, elbow=epositive, wrist=wpositive, fatherId=fReference[0]}
  [673] = {x=-361.301, y=104.782, z=198, rx=180, rz=114.796, shoulder=lefty, elbow=epositive, wrist=wpositive, fatherId=fReference[0]}
  [674] = {x=-348.732, y=131.989, z=198, rx=180, rz=124.454, shoulder=lefty, elbow=epositive, wrist=wpositive, fatherId=fReference[0]}
  [675] = {x=-331.776, y=156.702, z=198, rx=180, rz=134.113, shoulder=lefty, elbow=epositive, wrist=wpositive, fatherId=fReference[0]}
  [676] = {x=-310.915, y=178.22, z=198, rx=-180, rz=143.771, shoulder=lefty, elbow=epositive, wrist=wpositive, fatherId=fReference[0]}
  [677] = {x=-286.739, y=195.933, z=198, rx=180, rz=153.43, shoulder=lefty, elbow=epositive, wrist=wpositive, fatherId=fReference[0]}
  [678] = {x=-259.934, y=209.338, z=198, rx=180, rz=163.088, shoulder=lefty, elbow=epositive, wrist=wpositive, fatherId=fReference[0]}
  [679] = {x=-231.259, y=218.057, z=198, rx=180, rz=172.747, shoulder=lefty, elbow=epositive, wrist=wpositive, fatherId=fReference[0]}
  [680] = {x=-201.529, y=221.841, z=198, rx=-180, rz=179.696, shoulder=lefty, elbow=epositive, wrist=wpositive, fatherId=fReference[0]}
  [681] = {x=-171.525, y=222, z=198, rx=180, rz=-180, shoulder=lefty, elbow=epositive, wrist=wpositive, fatherId=fReference[0]}
  [682] = {x=-141.519, y=222, z=198, rx=180, rz=-180, shoulder=lefty, elbow=epositive, wrist=wpositive, fatherId=fReference[0]}
  [683] = {x=-111.513, y=222, z=198, rx=180, rz=-180, shoulder=lefty, elbow=epositive, wrist=wpositive, fatherId=fReference[0]}
  [684] = {x=-81.507, y=222, z=198, rx=-180, rz=-180, shoulder=lefty, elbow=epositive, wrist=wpositive, fatherId=fReference[0]}
  [685] = {x=-51.501, y=222, z=198, rx=-180, rz=-180, shoulder=lefty, elbow=epositive, wrist=wpositive, fatherId=fReference[0]}
  [686] = {x=-21.496, y=222, z=198, rx=-180, rz=-180, shoulder=lefty, elbow=epositive, wrist=wpositive, fatherId=fReference[0]}
  [687] = {x=8.51, y=222, z=198, rx=180, rz=-180, shoulder=lefty, elbow=epositive, wrist=wpositive, fatherId=fReference[0]}
  [688] = {x=38.516, y=222, z=198, rx=180, rz=-180, shoulder=lefty, elbow=epositive, wrist=wpositive, fatherId=fReference[0]}
  [689] = {x=68.522, y=222, z=198, rx=180, rz=-180, shoulder=lefty, elbow=epositive, wrist=wpositive, fatherId=fReference[0]}
  [690] = {x=98.528, y=222, z=198, rx=-180, rz=-180, shoulder=lefty, elbow=epositive, wrist=wpositive, fatherId=fReference[0]}
  [691] = {x=128.534, y=222, z=198, rx=-180, rz=-180, shoulder=lefty, elbow=epositive, wrist=wpositive, fatherId=fReference[0]}
  [692] = {x=158.54, y=222, z=198, rx=-180, rz=-180, shoulder=lefty, elbow=epositive, wrist=wpositive, fatherId=fReference[0]}
  [693] = {x=188.546, y=222, z=198, rx=180, rz=-176.767, shoulder=lefty, elbow=epositive, wrist=wpositive, fatherId=fReference[0]}
  [694] = {x=218.474, y=220.309, z=198, rx=180, rz=-167.268, shoulder=lefty, elbow=epositive, wrist=wpositive, fatherId=fReference[0]}
  [695] = {x=247.707, y=213.704, z=198, rx=-180, rz=-157.609, shoulder=lefty, elbow=epositive, wrist=wpositive, fatherId=fReference[0]}
  [696] = {x=275.418, y=202.288, z=198, rx=-180, rz=-147.951, shoulder=lefty, elbow=epositive, wrist=wpositive, fatherId=fReference[0]}
  [697] = {x=300.821, y=186.384, z=198, rx=-180, rz=-138.292, shoulder=lefty, elbow=epositive, wrist=wpositive, fatherId=fReference[0]}
  [698] = {x=323.195, y=166.444, z=198, rx=-180, rz=-128.634, shoulder=lefty, elbow=epositive, wrist=wpositive, fatherId=fReference[0]}
  [699] = {x=341.907, y=143.033, z=198, rx=-180, rz=-118.975, shoulder=lefty, elbow=epositive, wrist=wpositive, fatherId=fReference[0]}
  [700] = {x=356.426, y=116.814, z=198, rx=-180, rz=-109.317, shoulder=lefty, elbow=epositive, wrist=wpositive, fatherId=fReference[0]}
  [701] = {x=366.34, y=88.531, z=198, rx=-180, rz=-99.658, shoulder=lefty, elbow=epositive, wrist=wpositive, fatherId=fReference[0]}
  [702] = {x=371.368, y=58.985, z=198, rx=-180, rz=-91.207, shoulder=lefty, elbow=epositive, wrist=wpositive, fatherId=fReference[0]}
  [703] = {x=372, y=28.997, z=198, rx=-180, rz=-90, shoulder=lefty, elbow=epositive, wrist=wpositive, fatherId=fReference[0]}
  [704] = {x=372, y=-1.009, z=198, rx=180, rz=-90, shoulder=lefty, elbow=epositive, wrist=wpositive, fatherId=fReference[0]}
  [705] = {x=372, y=-31.015, z=198, rx=180, rz=-88.446, shoulder=lefty, elbow=epositive, wrist=wpositive, fatherId=fReference[0]}
  [706] = {x=371.187, y=-60.995, z=198, rx=180, rz=-79.692, shoulder=lefty, elbow=epositive, wrist=wpositive, fatherId=fReference[0]}
  [707] = {x=365.824, y=-90.481, z=198, rx=180, rz=-70.034, shoulder=lefty, elbow=epositive, wrist=wpositive, fatherId=fReference[0]}
  [708] = {x=355.59, y=-118.65, z=198, rx=180, rz=-60.375, shoulder=lefty, elbow=epositive, wrist=wpositive, fatherId=fReference[0]}
  [709] = {x=340.775, y=-144.703, z=198, rx=180, rz=-50.717, shoulder=lefty, elbow=epositive, wrist=wpositive, fatherId=fReference[0]}
  [710] = {x=321.799, y=-167.901, z=198, rx=-180, rz=-41.058, shoulder=lefty, elbow=epositive, wrist=wpositive, fatherId=fReference[0]}
  [711] = {x=299.2, y=-187.586, z=198, rx=-180, rz=-31.4, shoulder=lefty, elbow=epositive, wrist=wpositive, fatherId=fReference[0]}
  [712] = {x=273.619, y=-203.201, z=198, rx=180, rz=-21.741, shoulder=lefty, elbow=epositive, wrist=wpositive, fatherId=fReference[0]}
  [713] = {x=245.78, y=-214.302, z=198, rx=180, rz=-12.083, shoulder=lefty, elbow=epositive, wrist=wpositive, fatherId=fReference[0]}
  [714] = {x=216.474, y=-220.576, z=198, rx=-180, rz=-2.723, shoulder=lefty, elbow=epositive, wrist=wpositive, fatherId=fReference[0]}
  [715] = {x=186.528, y=-222, z=198, rx=-180, shoulder=lefty, elbow=epositive, wrist=wpositive, fatherId=fReference[0]}
  [716] = {x=156.522, y=-222, z=198, rx=180, shoulder=lefty, elbow=epositive, wrist=wpositive, fatherId=fReference[0]}
  [717] = {x=126.516, y=-222, z=198, rx=180, shoulder=lefty, elbow=epositive, wrist=wpositive, fatherId=fReference[0]}
  [718] = {x=96.51, y=-222, z=198, rx=-180, shoulder=lefty, elbow=epositive, wrist=wpositive, fatherId=fReference[0]}
  [719] = {x=66.504, y=-222, z=198, rx=180, shoulder=lefty, elbow=epositive, wrist=wpositive, fatherId=fReference[0]}
  [720] = {x=36.499, y=-222, z=198, rx=-180, shoulder=lefty, elbow=epositive, wrist=wpositive, fatherId=fReference[0]}
  [721] = {x=6.493, y=-222, z=198, rx=-180, shoulder=lefty, elbow=epositive, wrist=wpositive, fatherId=fReference[0]}
  [722] = {x=-23.513, y=-222, z=198, rx=180, shoulder=lefty, elbow=epositive, wrist=wpositive, fatherId=fReference[0]}
  [723] = {x=-53.519, y=-222, z=198, rx=180, shoulder=lefty, elbow=epositive, wrist=wpositive, fatherId=fReference[0]}
  [724] = {x=-83.525, y=-222, z=198, rx=-180, shoulder=lefty, elbow=epositive, wrist=wpositive, fatherId=fReference[0]}
  [725] = {x=-113.531, y=-222, z=198, rx=-180, shoulder=lefty, elbow=epositive, wrist=wpositive, fatherId=fReference[0]}
  [726] = {x=-143.537, y=-222, z=198, rx=-180, shoulder=lefty, elbow=epositive, wrist=wpositive, fatherId=fReference[0]}
  [727] = {x=-173.543, y=-222, z=198, rx=180, rz=0.489, shoulder=lefty, elbow=epositive, wrist=wpositive, fatherId=fReference[0]}
  [728] = {x=-203.544, y=-221.744, z=198, rx=180, rz=7.903, shoulder=lefty, elbow=epositive, wrist=wpositive, fatherId=fReference[0]}
  [729] = {x=-233.23, y=-217.623, z=198, rx=-180, rz=17.561, shoulder=lefty, elbow=epositive, wrist=wpositive, fatherId=fReference[0]}
  [730] = {x=-261.803, y=-208.58, z=198, rx=-180, rz=27.22, shoulder=lefty, elbow=epositive, wrist=wpositive, fatherId=fReference[0]}
  [731] = {x=-288.455, y=-194.872, z=198, rx=-180, rz=36.878, shoulder=lefty, elbow=epositive, wrist=wpositive, fatherId=fReference[0]}
  [732] = {x=-312.429, y=-176.886, z=198, rx=-180, rz=46.537, shoulder=lefty, elbow=epositive, wrist=wpositive, fatherId=fReference[0]}
  [733] = {x=-333.045, y=-155.133, z=198, rx=180, rz=56.195, shoulder=lefty, elbow=epositive, wrist=wpositive, fatherId=fReference[0]}
  [734] = {x=-349.719, y=-130.229, z=198, rx=-180, rz=65.854, shoulder=lefty, elbow=epositive, wrist=wpositive, fatherId=fReference[0]}
  [735] = {x=-361.979, y=-102.881, z=198, rx=-180, rz=75.512, shoulder=lefty, elbow=epositive, wrist=wpositive, fatherId=fReference[0]}
  [736] = {x=-369.477, y=-73.864, z=198, rx=-180, rz=85.171, shoulder=lefty, elbow=epositive, wrist=wpositive, fatherId=fReference[0]}
  [737] = {x=-372, y=-44, z=198, rx=-180, rz=85.171, shoulder=lefty, elbow=epositive, wrist=wpositive, fatherId=fReference[0]}
  [738] = {x=-372, y=-44, z=198, rx=-180, rz=85.171, shoulder=lefty, elbow=epositive, wrist=wpositive, fatherId=fReference[0]}
  [739] = {x=-372, y=-44, z=298, rx=-180, rz=85.171, shoulder=lefty, elbow=epositive, wrist=wpositive, fatherId=fReference[0]}
public tool tTool = {z=495, fatherId=flange[0], ioLink=valve1}
aio Tpompe = {link=CanIO\RemIO\remio0_QW}
dio doPompe = {link=CanIO\RemIO\remio0_Q}
dio doValve1 = {link=valve1}
dio doValve2 = {link=valve2}
num nTension = 3
num nTObtOpen = 6
num nTPompeOff
num nTPompeOn = 2
